KUKA KRL program: MyProgram_058().src

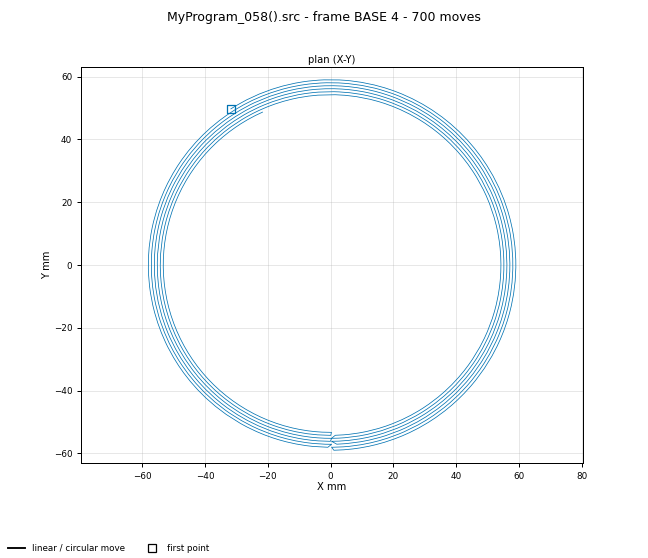
[picture p0: tool path of MyProgram_058().src in frame BASE 4, 700 of 700 moves have a stored position in this frame; points joined in program order, loops and branches not executed]
&ACCESS RVP
&REL 1
&PARAM TEMPLATE = C:\KRC\Roboter\Template\vorgabe
&PARAM EDITMASK = *
DEF MyProgram_058()
; ---- Setting reference (Base) ----
$BASE = BASE_DATA[4]

; --------------------------
; ---- Setting tool (TCP) ----
$TOOL = TOOL_DATA[3]
; --------------------------

$VEL.CP = VEL_APROX_PRINT
Startdeposition()
$VEL.CP = VEL_PRINT
LIN {X -31.7712,Y 49.7386,Z 70,A 115.7642,B 24.8628,C -2.7028,E1 24.9149,E2 -31.8987} C_DIS
LIN {X -30.2288,Y 50.6912,Z 70,A 113.4787,B 24.8635,C -2.6964,E1 24.9204,E2 -29.5909} C_DIS
LIN {X -26.7628,Y 52.603,Z 70,A 109.7045,B 24.8627,C -2.704,E1 24.9297,E2 -25.8244} C_DIS
LIN {X -22.7197,Y 54.4719,Z 70,A 105.0996,B 24.8626,C -2.7051,E1 24.9415,E2 -21.211} C_DIS
LIN {X -18.7389,Y 55.966,Z 70,A 100.782,B 24.8624,C -2.7067,E1 24.9529,E2 -16.8887} C_DIS
LIN {X -15.1635,Y 57.039,Z 70,A 97.4072,B 24.8616,C -2.7151,E1 24.9619,E2 -13.5286} C_DIS
LIN {X -11.2682,Y 57.9341,Z 70,A 94.0177,B 24.8603,C -2.7278,E1 24.9711,E2 -10.1653} C_DIS
LIN {X -8.899,Y 58.3451,Z 70,A 91.7622,B 24.8599,C -2.731,E1 24.9773,E2 -7.9152} C_DIS
LIN {X -6.9633,Y 58.6076,Z 70,A 89.5682,B 24.8604,C -2.7263,E1 24.9834,E2 -5.7084} C_DIS
LIN {X -3.7507,Y 58.9003,Z 70,A 86.8377,B 24.8595,C -2.7356,E1 24.9909,E2 -2.9988} C_DIS
LIN {X -2.0595,Y 58.9836,Z 70,A 84.3436,B 24.8611,C -2.7193,E1 24.998,E2 -0.4657} C_DIS
LIN {X 2.782,Y 58.9546,Z 70,A 80.395,B 24.8595,C -2.7349,E1 25.0089,E2 3.4453} C_DIS
LIN {X 4.6141,Y 58.8391,Z 70,A 78.6103,B 24.8595,C -2.7348,E1 25.0139,E2 5.2294} C_DIS
LIN {X 6.273,Y 58.6855,Z 70,A 76.5349,B 24.8605,C -2.7253,E1 25.0197,E2 7.326} C_DIS
LIN {X 9.7816,Y 58.2035,Z 70,A 73.055,B 24.8607,C -2.7235,E1 25.0293,E2 10.807} C_DIS
LIN {X 13.9156,Y 57.3558,Z 70,A 69.4123,B 24.8599,C -2.7308,E1 25.0392,E2 14.4274} C_DIS
LIN {X 17.2164,Y 56.4534,Z 70,A 65.518,B 24.8614,C -2.7167,E1 25.0497,E2 18.3487} C_DIS
LIN {X 20.0653,Y 55.5043,Z 70,A 63.2005,B 24.8604,C -2.7267,E1 25.0558,E2 20.6377} C_DIS
LIN {X 22.699,Y 54.4806,Z 70,A 59.2086,B 24.8633,C -2.6977,E1 25.0662,E2 24.6892} C_DIS
LIN {X 26.0309,Y 52.9694,Z 70,A 55.6174,B 24.8638,C -2.6926,E1 25.0752,E2 28.2831} C_DIS
LIN {X 29.3497,Y 51.2047,Z 70,A 52.1102,B 24.8641,C -2.6905,E1 25.0837,E2 31.7847} C_DIS
LIN {X 32.329,Y 49.3781,Z 70,A 49.9406,B 24.8619,C -2.7117,E1 25.0887,E2 33.8971} C_DIS
LIN {X 35.5242,Y 47.1314,Z 70,A 46.0197,B 24.8628,C -2.7025,E1 25.0976,E2 37.826} C_DIS
LIN {X 38.2213,Y 44.9718,Z 70,A 41.8696,B 24.8652,C -2.6788,E1 25.1066,E2 42.0164} C_DIS
LIN {X 40.951,Y 42.5011,Z 70,A 37.9748,B 24.8667,C -2.6645,E1 25.1145,E2 45.929} C_DIS
LIN {X 43.5029,Y 39.8852,Z 70,A 34.5086,B 24.8673,C -2.6586,E1 25.121,E2 49.3939} C_DIS
LIN {X 45.8007,Y 37.224,Z 70,A 32.1171,B 24.8658,C -2.6735,E1 25.1252,E2 51.7391} C_DIS
LIN {X 47.9004,Y 34.481,Z 70,A 29.1684,B 24.8657,C -2.6747,E1 25.1302,E2 54.671} C_DIS
LIN {X 49.7604,Y 31.7374,Z 70,A 25.887,B 24.8666,C -2.6651,E1 25.1353,E2 57.9586} C_DIS
LIN {X 51.7267,Y 28.4214,Z 70,A 22.1297,B 24.8676,C -2.655,E1 25.1406,E2 61.7206} C_DIS
LIN {X 53.6143,Y 24.6759,Z 70,A 17.7843,B 24.8694,C -2.6375,E1 25.146,E2 66.0841} C_DIS
LIN {X 55.207,Y 20.8685,Z 70,A 13.7674,B 24.8705,C -2.6259,E1 25.1502,E2 70.1063} C_DIS
LIN {X 56.4433,Y 17.2492,Z 70,A 10.1855,B 24.8713,C -2.618,E1 25.1533,E2 73.6865} C_DIS
LIN {X 57.2283,Y 14.428,Z 70,A 7.3114,B 24.8722,C -2.6088,E1 25.1554,E2 76.566} C_DIS
LIN {X 57.9039,Y 11.4254,Z 70,A 4.541,B 24.8726,C -2.6048,E1 25.157,E2 79.3297} C_DIS
LIN {X 58.3023,Y 9.1755,Z 70,A 1.1429,B 24.876,C -2.5705,E1 25.1585,E2 82.789} C_DIS
LIN {X 58.747,Y 5.6725,Z 70,A -0.9763,B 24.874,C -2.5903,E1 25.1591,E2 84.8487} C_DIS
LIN {X 58.9966,Y 1.6596,Z 70,A -5.4445,B 24.8765,C -2.5648,E1 25.1598,E2 89.3507} C_DIS
LIN {X 59.0156,Y -0.7643,Z 70,A -7.8914,B 24.8774,C -2.5551,E1 25.1598,E2 91.8058} C_DIS
LIN {X 58.8028,Y -5.0655,Z 70,A -11.3027,B 24.877,C -2.56,E1 25.1591,E2 95.1854} C_DIS
LIN {X 58.2932,Y -9.2343,Z 70,A -16.1939,B 24.88,C -2.528,E1 25.1573,E2 100.1234} C_DIS
LIN {X 57.5759,Y -12.9783,Z 70,A -19.3572,B 24.88,C -2.529,E1 25.1555,E2 103.266} C_DIS
LIN {X 57.0238,Y -15.2198,Z 70,A -21.3949,B 24.8801,C -2.5268,E1 25.1541,E2 105.297} C_DIS
LIN {X 56.2334,Y -17.922,Z 70,A -24.511,B 24.8818,C -2.5094,E1 25.1515,E2 108.4366} C_DIS
LIN {X 55.1794,Y -20.9418,Z 70,A -27.4296,B 24.8823,C -2.5043,E1 25.1487,E2 111.3509} C_DIS
LIN {X 54.1381,Y -23.5033,Z 70,A -30.0027,B 24.8828,C -2.4988,E1 25.146,E2 113.9226} C_DIS
LIN {X 53.029,Y -25.9104,Z 70,A -32.634,B 24.8836,C -2.4899,E1 25.1428,E2 116.561} C_DIS
LIN {X 51.3804,Y -29.0427,Z 70,A -35.9802,B 24.8844,C -2.4821,E1 25.1384,E2 119.9081} C_DIS
LIN {X 48.9651,Y -32.951,Z 70,A -40.4263,B 24.8855,C -2.47,E1 25.1317,E2 124.3604} C_DIS
LIN {X 46.171,Y -36.7642,Z 70,A -44.6881,B 24.8859,C -2.4653,E1 25.1246,E2 128.6128} C_DIS
LIN {X 44.7293,Y -38.506,Z 70,A -47.2824,B 24.8873,C -2.4505,E1 25.1199,E2 131.2303} C_DIS
LIN {X 42.5894,Y -40.8593,Z 70,A -50.345,B 24.8879,C -2.4435,E1 25.1141,E2 134.2961} C_DIS
LIN {X 40.4139,Y -43.0121,Z 70,A -53.3512,B 24.8887,C -2.4357,E1 25.108,E2 137.3082} C_DIS
LIN {X 38.5066,Y -44.7285,Z 70,A -55.5701,B 24.8887,C -2.4362,E1 25.1034,E2 139.517} C_DIS
LIN {X 36.3375,Y -46.5083,Z 70,A -59.4128,B 24.8914,C -2.4053,E1 25.0948,E2 143.4186} C_DIS
LIN {X 33.5039,Y -48.5887,Z 70,A -61.8182,B 24.89,C -2.4209,E1 25.0894,E2 145.7788} C_DIS
LIN {X 31.069,Y -50.1807,Z 70,A -64.8964,B 24.891,C -2.4099,E1 25.0821,E2 148.8731} C_DIS
LIN {X 28.1391,Y -51.8798,Z 70,A -68.1417,B 24.8914,C -2.4052,E1 25.0742,E2 152.1201} C_DIS
LIN {X 25.2158,Y -53.3627,Z 70,A -71.046,B 24.8914,C -2.4062,E1 25.067,E2 155.0143} C_DIS
LIN {X 22.836,Y -54.4229,Z 70,A -73.5731,B 24.8917,C -2.4025,E1 25.0605,E2 157.5439} C_DIS
LIN {X 20.2386,Y -55.4412,Z 70,A -76.3101,B 24.8921,C -2.3983,E1 25.0533,E2 160.285} C_DIS
LIN {X 17.1773,Y -56.4656,Z 70,A -79.6955,B 24.8929,C -2.3892,E1 25.0443,E2 163.6858} C_DIS
LIN {X 14.4326,Y -57.2285,Z 70,A -82.0061,B 24.8923,C -2.3961,E1 25.0381,E2 165.9764} C_DIS
LIN {X 12.2163,Y -57.7424,Z 70,A -84.4155,B 24.8928,C -2.3898,E1 25.0315,E2 168.3975} C_DIS
LIN {X 9.3879,Y -58.2693,Z 70,A -86.8704,B 24.8924,C -2.3948,E1 25.0248,E2 170.8379} C_DIS
LIN {X 7.1217,Y -58.5886,Z 70,A -89.4603,B 24.8932,C -2.3856,E1 25.0176,E2 173.4475} C_DIS
LIN {X 4.2204,Y -58.8691,Z 70,A -92.2877,B 24.8933,C -2.3843,E1 25.0097,E2 176.2766} C_DIS
LIN {X 1.0462,Y -59.0104,Z 70,A -95.2132,B 24.8931,C -2.3866,E1 25.0015,E2 179.196} C_DIS
LIN {X 1.0462,Y -59.0104,Z 70,A -95.2132,B 24.8931,C -2.3866,E1 25.0015,E2 179.196} C_DIS
Enddeposition()
LIN {X 0.3368,Y -58.0655,Z 70,A -95.8183,B 24.8915,C -2.4048,E1 25,E2 179.7576} C_DIS
Startdeposition()
$VEL.CP = VEL_PRINT
LIN {X 4.0061,Y -57.93,Z 70,A -91.3397,B 24.8898,C -2.4236,E1 25.0126,E2 175.2355} C_DIS
LIN {X 6.0336,Y -57.754,Z 70,A -88.5797,B 24.8882,C -2.4406,E1 25.0204,E2 172.437} C_DIS
LIN {X 9.6767,Y -57.2564,Z 70,A -84.9689,B 24.888,C -2.4428,E1 25.0303,E2 168.8244} C_DIS
LIN {X 12.7797,Y -56.6453,Z 70,A -82.2927,B 24.8886,C -2.436,E1 25.0376,E2 166.1679} C_DIS
LIN {X 15.542,Y -55.9504,Z 70,A -79.5466,B 24.8885,C -2.4375,E1 25.045,E2 163.4225} C_DIS
LIN {X 18.2311,Y -55.1325,Z 70,A -76.5661,B 24.8878,C -2.4453,E1 25.053,E2 160.4291} C_DIS
LIN {X 21.8468,Y -53.8019,Z 70,A -73.2635,B 24.8883,C -2.4395,E1 25.0615,E2 157.1474} C_DIS
LIN {X 23.4032,Y -53.1438,Z 70,A -70.8909,B 24.8866,C -2.4575,E1 25.0677,E2 154.7378} C_DIS
LIN {X 27.8224,Y -50.9692,Z 70,A -66.6091,B 24.8871,C -2.4526,E1 25.0783,E2 150.4795} C_DIS
LIN {X 30.5558,Y -49.3795,Z 70,A -63.1211,B 24.8858,C -2.4665,E1 25.0867,E2 146.9693} C_DIS
LIN {X 32.792,Y -47.9238,Z 70,A -60.5015,B 24.8854,C -2.4714,E1 25.0927,E2 144.3471} C_DIS
LIN {X 36.1303,Y -45.4594,Z 70,A -56.8016,B 24.8854,C -2.471,E1 25.1009,E2 140.6615} C_DIS
LIN {X 37.9818,Y -43.923,Z 70,A -54.0281,B 24.8841,C -2.4854,E1 25.1069,E2 137.8648} C_DIS
LIN {X 40.8451,Y -41.2748,Z 70,A -50.3062,B 24.8835,C -2.4915,E1 25.1144,E2 134.1438} C_DIS
LIN {X 43.5271,Y -38.435,Z 70,A -46.9008,B 24.8835,C -2.4907,E1 25.1208,E2 130.7553} C_DIS
LIN {X 45.0965,Y -36.5819,Z 70,A -43.953,B 24.8818,C -2.5096,E1 25.1261,E2 127.7763} C_DIS
LIN {X 47.5483,Y -33.3337,Z 70,A -40.6437,B 24.8823,C -2.504,E1 25.1315,E2 124.4963} C_DIS
LIN {X 48.9925,Y -31.1723,Z 70,A -37.4768,B 24.8803,C -2.5251,E1 25.1364,E2 121.2953} C_DIS
LIN {X 50.6871,Y -28.3328,Z 70,A -33.9859,B 24.8789,C -2.5398,E1 25.1412,E2 117.7878} C_DIS
LIN {X 52.8545,Y -24.0493,Z 70,A -30.051,B 24.8794,C -2.5348,E1 25.146,E2 113.8857} C_DIS
LIN {X 53.5161,Y -22.5379,Z 70,A -27.9151,B 24.8778,C -2.5516,E1 25.1484,E2 111.7218} C_DIS
LIN {X 54.8862,Y -18.9604,Z 70,A -24.4347,B 24.8774,C -2.556,E1 25.1517,E2 108.2504} C_DIS
LIN {X 55.7308,Y -16.3106,Z 70,A -21.7341,B 24.8766,C -2.5635,E1 25.1539,E2 105.5476} C_DIS
LIN {X 56.4512,Y -13.6094,Z 70,A -19.2381,B 24.8764,C -2.5659,E1 25.1556,E2 103.0603} C_DIS
LIN {X 57.3258,Y -9.2615,Z 70,A -14.9406,B 24.8753,C -2.5777,E1 25.1579,E2 98.7599} C_DIS
LIN {X 57.803,Y -5.5483,Z 70,A -11.1473,B 24.8739,C -2.5917,E1 25.1592,E2 94.956} C_DIS
LIN {X 58.0553,Y -1.2392,Z 70,A -6.9847,B 24.8728,C -2.6029,E1 25.1598,E2 90.7917} C_DIS
LIN {X 58.0291,Y 2.1446,Z 70,A -2.8172,B 24.8698,C -2.633,E1 25.1595,E2 86.5777} C_DIS
LIN {X 57.6965,Y 6.5634,Z 70,A 1.1575,B 24.8694,C -2.6372,E1 25.1584,E2 82.6167} C_DIS
LIN {X 57.2137,Y 9.9317,Z 70,A 4.1816,B 24.8692,C -2.6397,E1 25.1571,E2 79.6045} C_DIS
LIN {X 56.887,Y 11.653,Z 70,A 6.4002,B 24.8675,C -2.6565,E1 25.1559,E2 77.3591} C_DIS
LIN {X 55.7905,Y 16.1067,Z 70,A 10.1188,B 24.868,C -2.6511,E1 25.1533,E2 73.6746} C_DIS
LIN {X 54.7562,Y 19.3311,Z 70,A 13.5403,B 24.8669,C -2.6628,E1 25.1503,E2 70.2449} C_DIS
LIN {X 54.0939,Y 21.1138,Z 70,A 15.9706,B 24.865,C -2.6811,E1 25.1478,E2 67.7848} C_DIS
LIN {X 52.902,Y 23.9439,Z 70,A 19.526,B 24.8629,C -2.7018,E1 25.1437,E2 64.1997} C_DIS
LIN {X 51.104,Y 27.5739,Z 70,A 23.5816,B 24.8617,C -2.7139,E1 25.1384,E2 60.1368} C_DIS
LIN {X 49.4059,Y 30.5134,Z 70,A 25.7534,B 24.8636,C -2.6954,E1 25.1354,E2 58.02} C_DIS
LIN {X 47.5937,Y 33.2683,Z 70,A 29.4558,B 24.8617,C -2.7138,E1 25.1295,E2 54.2923} C_DIS
LIN {X 45.5686,Y 35.992,Z 70,A 32.214,B 24.8622,C -2.7083,E1 25.1249,E2 51.5601} C_DIS
LIN {X 43.7453,Y 38.1873,Z 70,A 35.3315,B 24.8609,C -2.7216,E1 25.1193,E2 48.4256} C_DIS
LIN {X 42.43,Y 39.6442,Z 70,A 38.0863,B 24.8586,C -2.7442,E1 25.1139,E2 45.6291} C_DIS
LIN {X 39.5187,Y 42.5478,Z 70,A 41.7521,B 24.8586,C -2.7436,E1 25.1065,E2 41.98} C_DIS
LIN {X 36.5071,Y 45.157,Z 70,A 45.3575,B 24.8586,C -2.7437,E1 25.0988,E2 38.3882} C_DIS
LIN {X 34.84,Y 46.4554,Z 70,A 47.519,B 24.8581,C -2.749,E1 25.094,E2 36.2219} C_DIS
LIN {X 31.8583,Y 48.5488,Z 70,A 50.6064,B 24.8586,C -2.7437,E1 25.087,E2 33.1575} C_DIS
LIN {X 28.6355,Y 50.5178,Z 70,A 55.493,B 24.8554,C -2.7743,E1 25.075,E2 28.2133} C_DIS
LIN {X 25.7741,Y 52.0348,Z 70,A 57.857,B 24.8569,C -2.7603,E1 25.0693,E2 25.889} C_DIS
LIN {X 21.8175,Y 53.8138,Z 70,A 61.9803,B 24.8568,C -2.7615,E1 25.0587,E2 21.7727} C_DIS
LIN {X 19.5455,Y 54.6808,Z 70,A 64.7617,B 24.8557,C -2.7717,E1 25.0514,E2 18.9729} C_DIS
LIN {X 15.6188,Y 55.928,Z 70,A 68.2352,B 24.8567,C -2.7623,E1 25.0422,E2 15.5279} C_DIS
LIN {X 14.1219,Y 56.3253,Z 70,A 70.4889,B 24.855,C -2.7783,E1 25.036,E2 13.2396} C_DIS
LIN {X 10.0125,Y 57.1992,Z 70,A 74.5226,B 24.855,C -2.7776,E1 25.0249,E2 9.2122} C_DIS
LIN {X 5.3929,Y 57.8173,Z 70,A 78.9116,B 24.8554,C -2.7741,E1 25.0128,E2 4.8347} C_DIS
LIN {X 2.5862,Y 58.0107,Z 70,A 81.7846,B 24.8553,C -2.776,E1 25.0048,E2 1.9583} C_DIS
LIN {X -1.2933,Y 58.0543,Z 70,A 85.1594,B 24.8563,C -2.7662,E1 24.9954,E2 -1.393} C_DIS
LIN {X -3.1849,Y 57.9809,Z 70,A 87.3647,B 24.8556,C -2.7722,E1 24.9892,E2 -3.6132} C_DIS
LIN {X -6.7659,Y 57.6728,Z 70,A 90.7348,B 24.8562,C -2.7669,E1 24.9799,E2 -6.9726} C_DIS
LIN {X -9.6106,Y 57.2675,Z 70,A 93.6963,B 24.8562,C -2.7675,E1 24.9717,E2 -9.938} C_DIS
LIN {X -12.5839,Y 56.6888,Z 70,A 96.8429,B 24.8561,C -2.768,E1 24.9631,E2 -13.0897} C_DIS
LIN {X -15.2568,Y 56.0283,Z 70,A 99.8798,B 24.8557,C -2.7715,E1 24.9549,E2 -16.1394} C_DIS
LIN {X -18.9545,Y 54.8884,Z 70,A 103.0395,B 24.8575,C -2.7545,E1 24.9466,E2 -19.2644} C_DIS
LIN {X -21.8103,Y 53.8168,Z 70,A 106.3993,B 24.8572,C -2.7571,E1 24.9378,E2 -22.6376} C_DIS
LIN {X -24.9043,Y 52.4574,Z 70,A 109.1655,B 24.8588,C -2.7416,E1 24.9308,E2 -25.3736} C_DIS
LIN {X -27.6387,Y 51.0689,Z 70,A 112.9934,B 24.8578,C -2.7515,E1 24.9213,E2 -29.2356} C_DIS
LIN {X -30.7549,Y 49.2551,Z 70,A 116.2345,B 24.8591,C -2.7393,E1 24.9136,E2 -32.4576} C_DIS
LIN {X -33.0294,Y 47.7599,Z 70,A 118.7367,B 24.8599,C -2.7308,E1 24.9078,E2 -34.9478} C_DIS
LIN {X -35.3908,Y 46.0372,Z 70,A 121.9748,B 24.8599,C -2.7313,E1 24.9005,E2 -38.1987} C_DIS
LIN {X -38.288,Y 43.6574,Z 70,A 125.3415,B 24.8613,C -2.7172,E1 24.8934,E2 -41.5448} C_DIS
LIN {X -40.5568,Y 41.5579,Z 70,A 128.7411,B 24.8614,C -2.7164,E1 24.8865,E2 -44.9565} C_DIS
LIN {X -42.9807,Y 39.0465,Z 70,A 132.2773,B 24.8621,C -2.7097,E1 24.8797,E2 -48.492} C_DIS
LIN {X -45.4039,Y 36.2004,Z 70,A 136.0486,B 24.8629,C -2.7017,E1 24.8731,E2 -52.2617} C_DIS
LIN {X -47.4887,Y 33.4194,Z 70,A 139.2387,B 24.8643,C -2.6883,E1 24.8679,E2 -55.4354} C_DIS
LIN {X -48.7906,Y 31.4868,Z 70,A 141.2399,B 24.8654,C -2.6769,E1 24.8648,E2 -57.4192} C_DIS
LIN {X -50.2196,Y 29.1544,Z 70,A 144.3862,B 24.8654,C -2.677,E1 24.8603,E2 -60.5821} C_DIS
LIN {X -51.8909,Y 26.063,Z 70,A 147.9848,B 24.8662,C -2.6693,E1 24.8557,E2 -64.1814} C_DIS
LIN {X -53.0729,Y 23.5646,Z 70,A 150.1524,B 24.868,C -2.6516,E1 24.8532,E2 -66.3187} C_DIS
LIN {X -54.2492,Y 20.7117,Z 70,A 154.0378,B 24.8674,C -2.6569,E1 24.8491,E2 -70.2385} C_DIS
LIN {X -55.4296,Y 17.3061,Z 70,A 157.3705,B 24.8689,C -2.6422,E1 24.8463,E2 -73.555} C_DIS
LIN {X -56.4076,Y 13.7882,Z 70,A 160.5004,B 24.8708,C -2.6229,E1 24.8441,E2 -76.6572} C_DIS
LIN {X -56.8516,Y 11.824,Z 70,A 162.5908,B 24.8713,C -2.6185,E1 24.8428,E2 -78.7492} C_DIS
LIN {X -57.2638,Y 9.6323,Z 70,A 165.1916,B 24.8713,C -2.6185,E1 24.8416,E2 -81.3653} C_DIS
LIN {X -57.8002,Y 5.5788,Z 70,A 169.254,B 24.8725,C -2.6061,E1 24.8403,E2 -85.4227} C_DIS
LIN {X -58.0131,Y 2.53,Z 70,A 172.2094,B 24.8735,C -2.5956,E1 24.8398,E2 -88.3706} C_DIS
LIN {X -58.0572,Y -1.1344,Z 70,A 175.4406,B 24.8753,C -2.5776,E1 24.8398,E2 -91.5783} C_DIS
LIN {X -57.982,Y -3.1649,Z 70,A 177.7382,B 24.8753,C -2.5763,E1 24.8401,E2 -93.8867} C_DIS
LIN {X -57.6791,Y -6.7118,Z 70,A -178.9542,B 24.8768,C -2.5619,E1 24.841,E2 -97.1795} C_DIS
LIN {X -57.3992,Y -8.7866,Z 70,A -176.0673,B 24.876,C -2.5697,E1 24.8422,E2 -100.1023} C_DIS
LIN {X -56.6399,Y -12.8033,Z 70,A -173.0126,B 24.8788,C -2.5405,E1 24.8439,E2 -103.1052} C_DIS
LIN {X -56.0504,Y -15.1747,Z 70,A -170.1321,B 24.8788,C -2.5413,E1 24.8459,E2 -106.0045} C_DIS
LIN {X -55.0664,Y -18.4267,Z 70,A -166.2436,B 24.8788,C -2.5408,E1 24.8493,E2 -109.9141} C_DIS
LIN {X -53.9363,Y -21.5135,Z 70,A -163.3509,B 24.8803,C -2.5254,E1 24.8522,E2 -112.7862} C_DIS
LIN {X -52.5831,Y -24.6365,Z 70,A -160.4693,B 24.882,C -2.5077,E1 24.8554,E2 -115.6413} C_DIS
LIN {X -51.8846,Y -26.0766,Z 70,A -158.2162,B 24.8812,C -2.5152,E1 24.8583,E2 -117.9245} C_DIS
LIN {X -50.001,Y -29.5262,Z 70,A -154.846,B 24.8831,C -2.496,E1 24.8629,E2 -121.2665} C_DIS
LIN {X -48.3842,Y -32.1081,Z 70,A -151.25,B 24.8828,C -2.4989,E1 24.8684,E2 -124.8875} C_DIS
LIN {X -46.7722,Y -34.4137,Z 70,A -148.7066,B 24.8838,C -2.488,E1 24.8725,E2 -127.4173} C_DIS
LIN {X -44.7315,Y -37.0274,Z 70,A -145.6423,B 24.8849,C -2.4767,E1 24.8779,E2 -130.4687} C_DIS
LIN {X -42.2486,Y -39.837,Z 70,A -141.3411,B 24.8846,C -2.4796,E1 24.886,E2 -134.7959} C_DIS
LIN {X -39.6939,Y -42.3832,Z 70,A -137.4422,B 24.8846,C -2.4787,E1 24.8939,E2 -138.7089} C_DIS
LIN {X -36.69,Y -45.0089,Z 70,A -133.4944,B 24.8853,C -2.4717,E1 24.9024,E2 -142.6549} C_DIS
LIN {X -33.2602,Y -47.5994,Z 70,A -129.5351,B 24.8865,C -2.4593,E1 24.9114,E2 -146.5985} C_DIS
LIN {X -28.6805,Y -50.4919,Z 70,A -124.9588,B 24.8886,C -2.4369,E1 24.9222,E2 -151.1355} C_DIS
LIN {X -26.639,Y -51.5979,Z 70,A -121.9747,B 24.8876,C -2.4473,E1 24.9296,E2 -154.1526} C_DIS
LIN {X -23.6199,Y -53.048,Z 70,A -119.1743,B 24.8888,C -2.4338,E1 24.9367,E2 -156.9279} C_DIS
LIN {X -21.0188,Y -54.131,Z 70,A -116.2578,B 24.8888,C -2.4338,E1 24.9442,E2 -159.8508} C_DIS
LIN {X -18.4558,Y -55.0574,Z 70,A -113.659,B 24.8892,C -2.4298,E1 24.9511,E2 -162.4452} C_DIS
LIN {X -16.2663,Y -55.744,Z 70,A -111.49,B 24.8895,C -2.4264,E1 24.9569,E2 -164.6096} C_DIS
LIN {X -14.0521,Y -56.3432,Z 70,A -109.1453,B 24.8895,C -2.4267,E1 24.9632,E2 -166.9585} C_DIS
LIN {X -11.0255,Y -57.012,Z 70,A -105.6761,B 24.8888,C -2.4337,E1 24.9728,E2 -170.4484} C_DIS
LIN {X -7.8663,Y -57.5333,Z 70,A -102.9456,B 24.8897,C -2.4242,E1 24.9802,E2 -173.1587} C_DIS
LIN {X -5.7466,Y -57.784,Z 70,A -100.2879,B 24.8887,C -2.4353,E1 24.9877,E2 -175.8443} C_DIS
LIN {X -0.8759,Y -58.0619,Z 70,A -95.9188,B 24.8895,C -2.4266,E1 24.9998,E2 -180.1935} C_DIS
LIN {X -0.8759,Y -58.0619,Z 70,A -95.9188,B 24.8895,C -2.4266,E1 24.9998,E2 -180.1935} C_DIS
Enddeposition()
LIN {X 0.3217,Y -57.1143,Z 70,A -94.8754,B 24.8882,C -2.4403,E1 25.0029,E2 -181.2696} C_DIS
Startdeposition()
$VEL.CP = VEL_PRINT
LIN {X -1.6753,Y -57.0923,Z 70,A -98.3895,B 24.891,C -2.4097,E1 24.9928,E2 -177.6824} C_DIS
LIN {X -5.5522,Y -56.8472,Z 70,A -101.9141,B 24.8904,C -2.417,E1 24.9831,E2 -174.1738} C_DIS
LIN {X -8.11,Y -56.5382,Z 70,A -104.2999,B 24.89,C -2.4214,E1 24.9765,E2 -171.7967} C_DIS
LIN {X -11.1706,Y -56.0141,Z 70,A -107.9954,B 24.8909,C -2.4113,E1 24.9663,E2 -168.0732} C_DIS
LIN {X -14.0088,Y -55.3725,Z 70,A -110.4419,B 24.8899,C -2.4218,E1 24.9597,E2 -165.6484} C_DIS
LIN {X -16.4763,Y -54.6884,Z 70,A -113.2493,B 24.8902,C -2.4189,E1 24.9521,E2 -162.8297} C_DIS
LIN {X -19.2701,Y -53.769,Z 70,A -116.3655,B 24.8902,C -2.4182,E1 24.9439,E2 -159.7057} C_DIS
LIN {X -22.8472,Y -52.3483,Z 70,A -119.8469,B 24.8893,C -2.4291,E1 24.9349,E2 -156.2425} C_DIS
LIN {X -24.9522,Y -51.3783,Z 70,A -122.9194,B 24.8903,C -2.4181,E1 24.9271,E2 -153.1358} C_DIS
LIN {X -28.4494,Y -49.5275,Z 70,A -126.7876,B 24.8896,C -2.4252,E1 24.9177,E2 -149.2735} C_DIS
LIN {X -32.168,Y -47.1967,Z 70,A -130.4275,B 24.8877,C -2.4457,E1 24.9092,E2 -145.6706} C_DIS
LIN {X -33.522,Y -46.2459,Z 70,A -133.1182,B 24.8892,C -2.43,E1 24.903,E2 -142.9332} C_DIS
LIN {X -36.8731,Y -43.6207,Z 70,A -137.4028,B 24.8885,C -2.4376,E1 24.8938,E2 -138.6504} C_DIS
LIN {X -40.1335,Y -40.6403,Z 70,A -141.4744,B 24.8871,C -2.4528,E1 24.8856,E2 -134.5982} C_DIS
LIN {X -42.9586,Y -37.6417,Z 70,A -145.4584,B 24.886,C -2.4644,E1 24.8781,E2 -130.6242} C_DIS
LIN {X -45.3182,Y -34.7651,Z 70,A -149.0744,B 24.885,C -2.4751,E1 24.8719,E2 -127.0168} C_DIS
LIN {X -47.3419,Y -31.9543,Z 70,A -152.4104,B 24.884,C -2.4859,E1 24.8665,E2 -123.6903} C_DIS
LIN {X -48.511,Y -30.1502,Z 70,A -154.7657,B 24.8838,C -2.4881,E1 24.863,E2 -121.3282} C_DIS
LIN {X -50.1157,Y -27.4004,Z 70,A -158.1128,B 24.8833,C -2.4939,E1 24.8584,E2 -117.9775} C_DIS
LIN {X -51.4173,Y -24.8721,Z 70,A -160.6434,B 24.882,C -2.5071,E1 24.8552,E2 -115.4647} C_DIS
LIN {X -52.8836,Y -21.5792,Z 70,A -164.253,B 24.8811,C -2.5173,E1 24.8512,E2 -111.8597} C_DIS
LIN {X -54.1577,Y -18.1463,Z 70,A -167.902,B 24.88,C -2.5283,E1 24.8478,E2 -108.2163} C_DIS
LIN {X -54.7147,Y -16.3909,Z 70,A -170.1922,B 24.8802,C -2.5265,E1 24.8459,E2 -105.9085} C_DIS
LIN {X -55.712,Y -12.5929,Z 70,A -173.6496,B 24.8783,C -2.5462,E1 24.8435,E2 -102.4781} C_DIS
LIN {X -56.1934,Y -10.2262,Z 70,A -176.5738,B 24.8783,C -2.5454,E1 24.842,E2 -99.5348} C_DIS
LIN {X -56.6922,Y -6.9596,Z 70,A -179.8253,B 24.8773,C -2.5567,E1 24.8407,E2 -96.2907} C_DIS
LIN {X -56.9947,Y -3.736,Z 70,A 177.283,B 24.8757,C -2.5726,E1 24.8401,E2 -93.4198} C_DIS
LIN {X -57.0847,Y -1.9147,Z 70,A 174.667,B 24.8764,C -2.5656,E1 24.8398,E2 -90.7713} C_DIS
LIN {X -57.0521,Y 2.7317,Z 70,A 170.6679,B 24.874,C -2.591,E1 24.84,E2 -86.8089} C_DIS
LIN {X -56.9354,Y 4.5496,Z 70,A 168.7831,B 24.8735,C -2.5959,E1 24.8404,E2 -84.9244} C_DIS
LIN {X -56.7303,Y 6.6343,Z 70,A 166.4728,B 24.8732,C -2.5991,E1 24.8411,E2 -82.608} C_DIS
LIN {X -56.3312,Y 9.4407,Z 70,A 163.9146,B 24.8718,C -2.6127,E1 24.8422,E2 -80.0669} C_DIS
LIN {X -56.0575,Y 10.9505,Z 70,A 162.0738,B 24.8718,C -2.6126,E1 24.8431,E2 -78.215} C_DIS
LIN {X -55.475,Y 13.5966,Z 70,A 159.2999,B 24.8711,C -2.6201,E1 24.8449,E2 -75.4429} C_DIS
LIN {X -54.692,Y 16.4675,Z 70,A 156.3825,B 24.8701,C -2.6305,E1 24.8471,E2 -72.5332} C_DIS
LIN {X -53.5452,Y 19.8799,Z 70,A 152.7682,B 24.869,C -2.6414,E1 24.8504,E2 -68.9246} C_DIS
LIN {X -52.6274,Y 22.1968,Z 70,A 150.2278,B 24.8683,C -2.6482,E1 24.8531,E2 -66.3864} C_DIS
LIN {X -51.6026,Y 24.4848,Z 70,A 147.6106,B 24.8677,C -2.6539,E1 24.8562,E2 -63.7685} C_DIS
LIN {X -50.3353,Y 26.9957,Z 70,A 144.3789,B 24.8677,C -2.6553,E1 24.8604,E2 -60.5229} C_DIS
LIN {X -47.9485,Y 31.0375,Z 70,A 140.3994,B 24.8651,C -2.6806,E1 24.8661,E2 -56.5833} C_DIS
LIN {X -46.9904,Y 32.4694,Z 70,A 138.1496,B 24.8655,C -2.6766,E1 24.8697,E2 -54.3128} C_DIS
LIN {X -44.6391,Y 35.6337,Z 70,A 133.5561,B 24.8655,C -2.6763,E1 24.8776,E2 -49.697} C_DIS
LIN {X -41.9452,Y 38.7682,Z 70,A 130.239,B 24.863,C -2.7005,E1 24.8836,E2 -46.4227} C_DIS
LIN {X -40.251,Y 40.5243,Z 70,A 127.7415,B 24.8625,C -2.7055,E1 24.8885,E2 -43.9265} C_DIS
LIN {X -37.922,Y 42.7119,Z 70,A 124.8382,B 24.8613,C -2.7179,E1 24.8945,E2 -41.0412} C_DIS
LIN {X -36.0728,Y 44.2844,Z 70,A 121.9721,B 24.8615,C -2.7158,E1 24.9006,E2 -38.159} C_DIS
LIN {X -34.1636,Y 45.7735,Z 70,A 119.7642,B 24.8606,C -2.7246,E1 24.9055,E2 -35.9642} C_DIS
LIN {X -32.2973,Y 47.1083,Z 70,A 116.9257,B 24.8611,C -2.7199,E1 24.9121,E2 -33.1046} C_DIS
LIN {X -28.9029,Y 49.2645,Z 70,A 113.029,B 24.8601,C -2.7295,E1 24.9213,E2 -29.2189} C_DIS
LIN {X -25.5964,Y 51.061,Z 70,A 109.711,B 24.8586,C -2.7438,E1 24.9294,E2 -25.9258} C_DIS
LIN {X -24.2242,Y 51.7256,Z 70,A 107.3219,B 24.8599,C -2.7309,E1 24.9356,E2 -23.4999} C_DIS
LIN {X -19.252,Y 53.7755,Z 70,A 101.9478,B 24.8592,C -2.7384,E1 24.9496,E2 -18.1321} C_DIS
LIN {X -15.0599,Y 55.0959,Z 70,A 98.327,B 24.8572,C -2.7575,E1 24.9591,E2 -14.5508} C_DIS
LIN {X -13.439,Y 55.5134,Z 70,A 96.3859,B 24.8575,C -2.7543,E1 24.9644,E2 -12.5993} C_DIS
LIN {X -10.8751,Y 56.072,Z 70,A 93.5266,B 24.8577,C -2.7522,E1 24.9723,E2 -9.7318} C_DIS
LIN {X -6.992,Y 56.6884,Z 70,A 89.8684,B 24.8569,C -2.7601,E1 24.9823,E2 -6.0893} C_DIS
LIN {X -4.5327,Y 56.9367,Z 70,A 87.4552,B 24.8567,C -2.7626,E1 24.989,E2 -3.6808} C_DIS
LIN {X -1.944,Y 57.0841,Z 70,A 84.6806,B 24.8569,C -2.7601,E1 24.9968,E2 -0.8998} C_DIS
LIN {X 0.909,Y 57.1098,Z 70,A 81.7964,B 24.8569,C -2.7602,E1 25.0048,E2 1.984} C_DIS
LIN {X 3.3817,Y 57.0171,Z 70,A 79.4695,B 24.8566,C -2.7633,E1 25.0113,E2 4.3028} C_DIS
LIN {X 5.6615,Y 56.8363,Z 70,A 77.1417,B 24.8566,C -2.7625,E1 25.0178,E2 6.6313} C_DIS
LIN {X 8.6238,Y 56.4622,Z 70,A 73.9556,B 24.8571,C -2.758,E1 25.0266,E2 9.8252} C_DIS
LIN {X 11.722,Y 55.9016,Z 70,A 70.7921,B 24.8573,C -2.7566,E1 25.0353,E2 12.9883} C_DIS
LIN {X 14.1408,Y 55.3388,Z 70,A 68.6854,B 24.8566,C -2.7629,E1 25.041,E2 15.077} C_DIS
LIN {X 16.245,Y 54.758,Z 70,A 66.3068,B 24.8572,C -2.7576,E1 25.0474,E2 17.4642} C_DIS
LIN {X 18.5443,Y 54.0231,Z 70,A 63.8601,B 24.8574,C -2.7551,E1 25.0538,E2 19.912} C_DIS
LIN {X 21.02,Y 53.1085,Z 70,A 61.0514,B 24.858,C -2.7494,E1 25.0612,E2 22.7284} C_DIS
LIN {X 25.3508,Y 51.1827,Z 70,A 57.0895,B 24.8569,C -2.7604,E1 25.0712,E2 26.6542} C_DIS
LIN {X 27.9188,Y 49.8285,Z 70,A 53.0381,B 24.8597,C -2.7328,E1 25.0813,E2 30.7593} C_DIS
LIN {X 31.1722,Y 47.8615,Z 70,A 49.698,B 24.8593,C -2.737,E1 25.0891,E2 34.0789} C_DIS
LIN {X 33.6583,Y 46.1462,Z 70,A 46.7534,B 24.8596,C -2.7337,E1 25.0958,E2 37.021} C_DIS
LIN {X 36.0869,Y 44.273,Z 70,A 43.6021,B 24.8604,C -2.7266,E1 25.1027,E2 40.1774} C_DIS
LIN {X 38.6321,Y 42.0702,Z 70,A 40.356,B 24.8608,C -2.7229,E1 25.1095,E2 43.4195} C_DIS
LIN {X 41.3505,Y 39.4017,Z 70,A 36.5769,B 24.8615,C -2.7158,E1 25.117,E2 47.1993} C_DIS
LIN {X 43.9326,Y 36.5001,Z 70,A 32.8699,B 24.862,C -2.7112,E1 25.1238,E2 50.9005} C_DIS
LIN {X 45.0415,Y 35.1236,Z 70,A 30.629,B 24.8634,C -2.6968,E1 25.1277,E2 53.165} C_DIS
LIN {X 47.0762,Y 32.3449,Z 70,A 27.132,B 24.8644,C -2.6874,E1 25.1333,E2 56.6672} C_DIS
LIN {X 48.7104,Y 29.8273,Z 70,A 23.7598,B 24.866,C -2.6717,E1 25.1383,E2 60.0594} C_DIS
LIN {X 51.2874,Y 25.1376,Z 70,A 18.755,B 24.8666,C -2.6653,E1 25.1448,E2 65.053} C_DIS
LIN {X 52.3557,Y 22.8303,Z 70,A 16.4453,B 24.8668,C -2.6635,E1 25.1474,E2 67.3543} C_DIS
LIN {X 53.7973,Y 19.1905,Z 70,A 12.6312,B 24.8677,C -2.6547,E1 25.1512,E2 71.1679} C_DIS
LIN {X 54.6598,Y 16.575,Z 70,A 10.1111,B 24.8679,C -2.6521,E1 25.1533,E2 73.68} C_DIS
LIN {X 55.4234,Y 13.8079,Z 70,A 6.7547,B 24.8699,C -2.6327,E1 25.1557,E2 77.063} C_DIS
LIN {X 56.0433,Y 11.0241,Z 70,A 4.3528,B 24.8697,C -2.6343,E1 25.1571,E2 79.4469} C_DIS
LIN {X 56.4592,Y 8.643,Z 70,A 1.8552,B 24.8706,C -2.6252,E1 25.1582,E2 81.9515} C_DIS
LIN {X 56.9311,Y 4.6027,Z 70,A -2.5882,B 24.8727,C -2.6043,E1 25.1595,E2 86.418} C_DIS
LIN {X 57.1153,Y 0.5249,Z 70,A -6.1775,B 24.8727,C -2.6029,E1 25.1598,E2 89.9893} C_DIS
LIN {X 57.0817,Y -2.0223,Z 70,A -9.2435,B 24.8747,C -2.5832,E1 25.1595,E2 93.0836} C_DIS
LIN {X 56.8278,Y -5.7427,Z 70,A -13.1144,B 24.8762,C -2.5684,E1 25.1586,E2 96.9665} C_DIS
LIN {X 56.3932,Y -9.0699,Z 70,A -17.0409,B 24.8784,C -2.5452,E1 25.1569,E2 100.9249} C_DIS
LIN {X 55.6853,Y -12.7084,Z 70,A -19.1599,B 24.876,C -2.5698,E1 25.1557,E2 102.9733} C_DIS
LIN {X 55.3353,Y -14.1543,Z 70,A -21.5989,B 24.8785,C -2.5436,E1 25.154,E2 105.4602} C_DIS
LIN {X 54.389,Y -17.4411,Z 70,A -24.2849,B 24.8779,C -2.5499,E1 25.1518,E2 108.1159} C_DIS
LIN {X 53.3253,Y -20.4649,Z 70,A -28.2362,B 24.8805,C -2.5235,E1 25.1479,E2 112.1077} C_DIS
LIN {X 52.1008,Y -23.4061,Z 70,A -31.2725,B 24.881,C -2.5175,E1 25.1445,E2 115.1414} C_DIS
LIN {X 49.8399,Y -27.8985,Z 70,A -35.9714,B 24.8817,C -2.5107,E1 25.1385,E2 119.8316} C_DIS
LIN {X 48.0818,Y -30.8298,Z 70,A -39.6105,B 24.883,C -2.4964,E1 25.1331,E2 123.4861} C_DIS
LIN {X 45.476,Y -34.5597,Z 70,A -44.3078,B 24.8844,C -2.4812,E1 25.1253,E2 128.1966} C_DIS
LIN {X 43.3292,Y -37.2151,Z 70,A -47.8088,B 24.8854,C -2.4708,E1 25.119,E2 131.7063} C_DIS
LIN {X 40.1677,Y -40.6065,Z 70,A -52.2194,B 24.886,C -2.4648,E1 25.1105,E2 136.1121} C_DIS
LIN {X 36.7463,Y -43.728,Z 70,A -56.3797,B 24.886,C -2.465,E1 25.1018,E2 140.2555} C_DIS
LIN {X 34.02,Y -45.8813,Z 70,A -60.4545,B 24.8878,C -2.4448,E1 25.0927,E2 144.3631} C_DIS
LIN {X 30.2725,Y -48.4346,Z 70,A -64.7283,B 24.8881,C -2.442,E1 25.0827,E2 148.6295} C_DIS
LIN {X 27.6275,Y -49.9912,Z 70,A -68.4137,B 24.8897,C -2.4238,E1 25.0737,E2 152.3473} C_DIS
LIN {X 23.8797,Y -51.886,Z 70,A -71.705,B 24.8886,C -2.4366,E1 25.0655,E2 155.5995} C_DIS
LIN {X 22.0826,Y -52.6754,Z 70,A -74.2462,B 24.8899,C -2.4217,E1 25.0589,E2 158.17} C_DIS
LIN {X 17.5486,Y -54.3542,Z 70,A -78.2924,B 24.889,C -2.4324,E1 25.0483,E2 162.1826} C_DIS
LIN {X 15.7517,Y -54.9022,Z 70,A -80.9348,B 24.8906,C -2.4146,E1 25.0411,E2 164.8628} C_DIS
LIN {X 12.341,Y -55.768,Z 70,A -84.4523,B 24.8909,C -2.4116,E1 25.0315,E2 168.3827} C_DIS
LIN {X 9.5701,Y -56.3096,Z 70,A -86.7919,B 24.8901,C -2.4194,E1 25.0252,E2 170.7012} C_DIS
LIN {X 4.9251,Y -56.9037,Z 70,A -91.3339,B 24.8901,C -2.4198,E1 25.0126,E2 175.2389} C_DIS
LIN {X 1.9775,Y -57.0831,Z 70,A -93.9877,B 24.8897,C -2.4248,E1 25.0052,E2 177.8798} C_DIS
LIN {X 1.9775,Y -57.0831,Z 70,A -93.9877,B 24.8897,C -2.4248,E1 25.0052,E2 177.8798} C_DIS
Enddeposition()
LIN {X 0.3099,Y -56.1615,Z 70,A -95.1001,B 24.8872,C -2.4521,E1 25.0023,E2 178.9272} C_DIS
Startdeposition()
$VEL.CP = VEL_PRINT
LIN {X 2.6789,Y -56.1021,Z 70,A -92.4847,B 24.8867,C -2.4568,E1 25.0096,E2 176.3012} C_DIS
LIN {X 5.8531,Y -55.8596,Z 70,A -88.772,B 24.8857,C -2.4679,E1 25.02,E2 172.5642} C_DIS
LIN {X 9.423,Y -55.3696,Z 70,A -85.7766,B 24.8867,C -2.4565,E1 25.0282,E2 169.5987} C_DIS
LIN {X 12.0412,Y -54.8596,Z 70,A -82.7636,B 24.886,C -2.4649,E1 25.0365,E2 166.5696} C_DIS
LIN {X 14.7486,Y -54.1943,Z 70,A -79.98,B 24.8858,C -2.4665,E1 25.044,E2 163.7865} C_DIS
LIN {X 16.8646,Y -53.5743,Z 70,A -77.2278,B 24.8846,C -2.4797,E1 25.0514,E2 161.008} C_DIS
LIN {X 21.2307,Y -51.9983,Z 70,A -72.9884,B 24.885,C -2.4755,E1 25.0624,E2 156.7878} C_DIS
LIN {X 24.6249,Y -50.4805,Z 70,A -68.5583,B 24.8832,C -2.495,E1 25.0737,E2 152.3227} C_DIS
LIN {X 28.1829,Y -48.5833,Z 70,A -65.3462,B 24.8843,C -2.4826,E1 25.0815,E2 149.1493} C_DIS
LIN {X 30.3057,Y -47.2876,Z 70,A -62.5744,B 24.8834,C -2.4924,E1 25.0881,E2 146.3631} C_DIS
LIN {X 33.2374,Y -45.2751,Z 70,A -58.3058,B 24.8814,C -2.5138,E1 25.0979,E2 142.0588} C_DIS
LIN {X 35.8999,Y -43.1944,Z 70,A -54.8107,B 24.8806,C -2.5224,E1 25.1054,E2 138.5567} C_DIS
LIN {X 38.7408,Y -40.6668,Z 70,A -51.7682,B 24.8815,C -2.5127,E1 25.1116,E2 135.5495} C_DIS
LIN {X 40.1793,Y -39.2462,Z 70,A -49.7464,B 24.8811,C -2.5167,E1 25.1156,E2 133.5267} C_DIS
LIN {X 42.9785,Y -36.1596,Z 70,A -45.7047,B 24.8805,C -2.5227,E1 25.1231,E2 129.4889} C_DIS
LIN {X 44.8828,Y -33.7653,Z 70,A -41.8604,B 24.8782,C -2.5472,E1 25.1297,E2 125.605} C_DIS
LIN {X 46.9702,Y -30.7957,Z 70,A -38.4862,B 24.8779,C -2.5498,E1 25.135,E2 122.2411} C_DIS
LIN {X 48.9813,Y -27.4845,Z 70,A -34.9648,B 24.8779,C -2.5513,E1 25.14,E2 118.7343} C_DIS
LIN {X 50.3208,Y -24.9475,Z 70,A -31.2779,B 24.8753,C -2.5771,E1 25.1447,E2 115.006} C_DIS
LIN {X 51.7186,Y -21.9016,Z 70,A -27.9155,B 24.8744,C -2.586,E1 25.1484,E2 111.6409} C_DIS
LIN {X 53.3277,Y -17.6302,Z 70,A -23.8813,B 24.8744,C -2.5859,E1 25.1522,E2 107.6296} C_DIS
LIN {X 53.9899,Y -15.4816,Z 70,A -20.9183,B 24.8723,C -2.6083,E1 25.1546,E2 104.6304} C_DIS
LIN {X 54.7862,Y -12.3734,Z 70,A -18.4543,B 24.8731,C -2.6,E1 25.1561,E2 102.2005} C_DIS
LIN {X 55.4601,Y -8.8781,Z 70,A -14.6993,B 24.8717,C -2.6142,E1 25.158,E2 98.4338} C_DIS
LIN {X 55.8508,Y -5.9375,Z 70,A -11.1978,B 24.8697,C -2.6347,E1 25.1592,E2 94.9046} C_DIS
LIN {X 56.1091,Y -2.5166,Z 70,A -8.197,B 24.8697,C -2.6343,E1 25.1597,E2 91.9225} C_DIS
LIN {X 56.1668,Y 0.2,Z 70,A -5.4342,B 24.8689,C -2.6428,E1 25.1597,E2 89.1561} C_DIS
LIN {X 55.9905,Y 4.4293,Z 70,A -0.637,B 24.8664,C -2.6673,E1 25.159,E2 84.3293} C_DIS
LIN {X 55.5762,Y 8.117,Z 70,A 2.6392,B 24.8664,C -2.6673,E1 25.1578,E2 81.0724} C_DIS
LIN {X 55.1477,Y 10.6439,Z 70,A 5.3354,B 24.8654,C -2.6773,E1 25.1565,E2 78.3686} C_DIS
LIN {X 54.4955,Y 13.5963,Z 70,A 8.3622,B 24.8646,C -2.6853,E1 25.1545,E2 75.3404} C_DIS
LIN {X 53.8757,Y 15.8736,Z 70,A 10.5349,B 24.8644,C -2.6871,E1 25.1529,E2 73.1757} C_DIS
LIN {X 52.9179,Y 18.823,Z 70,A 13.7862,B 24.8633,C -2.6984,E1 25.15,E2 69.9162} C_DIS
LIN {X 51.8421,Y 21.6098,Z 70,A 16.7159,B 24.8626,C -2.7044,E1 25.147,E2 66.9884} C_DIS
LIN {X 51.0557,Y 23.406,Z 70,A 19.1705,B 24.861,C -2.7202,E1 25.1441,E2 64.5098} C_DIS
LIN {X 49.1752,Y 27.1373,Z 70,A 23.6062,B 24.8595,C -2.7355,E1 25.1383,E2 60.0612} C_DIS
LIN {X 47.3732,Y 30.1724,Z 70,A 26.7801,B 24.8595,C -2.7353,E1 25.1337,E2 56.904} C_DIS
LIN {X 45.4429,Y 33.0082,Z 70,A 30.6803,B 24.8577,C -2.7528,E1 25.1274,E2 52.9815} C_DIS
LIN {X 43.4292,Y 35.6169,Z 70,A 33.6442,B 24.8577,C -2.7518,E1 25.1222,E2 50.0336} C_DIS
LIN {X 41.4927,Y 37.8542,Z 70,A 36.3135,B 24.8579,C -2.7509,E1 25.1173,E2 47.3784} C_DIS
LIN {X 40.2651,Y 39.1579,Z 70,A 38.7349,B 24.8561,C -2.7677,E1 25.1125,E2 44.9276} C_DIS
LIN {X 37.7454,Y 41.5925,Z 70,A 41.9199,B 24.8562,C -2.7665,E1 25.1061,E2 41.7586} C_DIS
LIN {X 35.4125,Y 43.5949,Z 70,A 45.3599,B 24.855,C -2.7788,E1 25.0987,E2 38.3025} C_DIS
LIN {X 32.7378,Y 45.6378,Z 70,A 49.1179,B 24.8536,C -2.7916,E1 25.0901,E2 34.5275} C_DIS
LIN {X 29.6916,Y 47.6757,Z 70,A 52.0111,B 24.8549,C -2.7795,E1 25.0834,E2 31.6725} C_DIS
LIN {X 27.202,Y 49.1391,Z 70,A 55.5159,B 24.8532,C -2.7953,E1 25.0749,E2 28.1408} C_DIS
LIN {X 22.8159,Y 51.3232,Z 70,A 60.5747,B 24.8525,C -2.8023,E1 25.0621,E2 23.0782} C_DIS
LIN {X 19.4788,Y 52.68,Z 70,A 64.2815,B 24.852,C -2.8064,E1 25.0524,E2 19.3697} C_DIS
LIN {X 15.2101,Y 54.0668,Z 70,A 68.3294,B 24.8528,C -2.799,E1 25.0417,E2 15.3467} C_DIS
LIN {X 12.5261,Y 54.751,Z 70,A 70.9939,B 24.853,C -2.7973,E1 25.0345,E2 12.69} C_DIS
LIN {X 10.4767,Y 55.1798,Z 70,A 73.2347,B 24.8527,C -2.8003,E1 25.0283,E2 10.4448} C_DIS
LIN {X 8.1113,Y 55.5771,Z 70,A 75.6281,B 24.8527,C -2.8,E1 25.0217,E2 8.0544} C_DIS
LIN {X 5.8868,Y 55.8561,Z 70,A 77.8801,B 24.8527,C -2.7997,E1 25.0155,E2 5.8048} C_DIS
LIN {X 3.6015,Y 56.0501,Z 70,A 80.3885,B 24.8524,C -2.8031,E1 25.0085,E2 3.2896} C_DIS
LIN {X 1.173,Y 56.1534,Z 70,A 82.6468,B 24.8529,C -2.7986,E1 25.0022,E2 1.0426} C_DIS
LIN {X -1.7021,Y 56.1396,Z 70,A 86.0437,B 24.852,C -2.8068,E1 24.9927,E2 -2.374} C_DIS
LIN {X -4.7622,Y 55.9635,Z 70,A 88.9173,B 24.8527,C -2.8006,E1 24.9847,E2 -5.2341} C_DIS
LIN {X -6.9618,Y 55.7324,Z 70,A 91.4628,B 24.8522,C -2.8048,E1 24.9776,E2 -7.7913} C_DIS
LIN {X -10.6785,Y 55.141,Z 70,A 94.7694,B 24.8536,C -2.792,E1 24.9686,E2 -11.0708} C_DIS
LIN {X -12.5666,Y 54.7416,Z 70,A 96.8936,B 24.8534,C -2.7932,E1 24.9628,E2 -13.2004} C_DIS
LIN {X -14.8631,Y 54.1636,Z 70,A 99.3128,B 24.8537,C -2.7909,E1 24.9563,E2 -15.6177} C_DIS
LIN {X -17.0677,Y 53.5096,Z 70,A 101.9025,B 24.8535,C -2.7927,E1 24.9493,E2 -18.2163} C_DIS
LIN {X -19.8913,Y 52.5252,Z 70,A 104.6064,B 24.8546,C -2.7826,E1 24.9423,E2 -20.9015} C_DIS
LIN {X -22.2843,Y 51.5558,Z 70,A 107.4815,B 24.8545,C -2.7833,E1 24.9348,E2 -23.7848} C_DIS
LIN {X -24.684,Y 50.4514,Z 70,A 110.1514,B 24.855,C -2.7787,E1 24.9281,E2 -26.4505} C_DIS
LIN {X -27.0913,Y 49.2003,Z 70,A 112.924,B 24.8554,C -2.7742,E1 24.9213,E2 -29.2202} C_DIS
LIN {X -30.2596,Y 47.3168,Z 70,A 117.4904,B 24.8547,C -2.7816,E1 24.9104,E2 -33.8186} C_DIS
LIN {X -32.8585,Y 45.5517,Z 70,A 120.4546,B 24.8558,C -2.771,E1 24.9037,E2 -36.7677} C_DIS
LIN {X -36.7933,Y 42.4364,Z 70,A 124.9197,B 24.8581,C -2.7486,E1 24.8941,E2 -41.1963} C_DIS
LIN {X -39.6173,Y 39.8129,Z 70,A 128.9784,B 24.8588,C -2.7417,E1 24.8859,E2 -45.2551} C_DIS
LIN {X -41.1951,Y 38.1785,Z 70,A 131.6426,B 24.8588,C -2.7419,E1 24.8808,E2 -47.9316} C_DIS
LIN {X -43.8885,Y 35.049,Z 70,A 135.2307,B 24.861,C -2.7207,E1 24.8744,E2 -51.4855} C_DIS
LIN {X -45.3926,Y 33.077,Z 70,A 138.6657,B 24.8601,C -2.7292,E1 24.8686,E2 -54.9573} C_DIS
LIN {X -47.386,Y 30.1517,Z 70,A 142.246,B 24.8612,C -2.7188,E1 24.8632,E2 -58.5307} C_DIS
LIN {X -49.6077,Y 26.3376,Z 70,A 146.1276,B 24.8635,C -2.6957,E1 24.8579,E2 -62.3774} C_DIS
LIN {X -50.4427,Y 24.6998,Z 70,A 148.3114,B 24.8635,C -2.6953,E1 24.8552,E2 -64.572} C_DIS
LIN {X -51.8803,Y 21.5196,Z 70,A 152.1328,B 24.8642,C -2.689,E1 24.8509,E2 -68.3995} C_DIS
LIN {X -53.3851,Y 17.4532,Z 70,A 156.3071,B 24.866,C -2.6715,E1 24.8471,E2 -72.5556} C_DIS
LIN {X -54.0402,Y 15.3041,Z 70,A 158.9314,B 24.8661,C -2.6699,E1 24.8451,E2 -75.1912} C_DIS
LIN {X -54.7701,Y 12.4406,Z 70,A 162.1172,B 24.8668,C -2.6633,E1 24.843,E2 -78.38} C_DIS
LIN {X -55.3987,Y 9.2491,Z 70,A 165.0301,B 24.8685,C -2.6462,E1 24.8416,E2 -81.2694} C_DIS
LIN {X -55.8623,Y 5.8274,Z 70,A 168.8128,B 24.8692,C -2.6394,E1 24.8404,E2 -85.0584} C_DIS
LIN {X -56.089,Y 2.9338,Z 70,A 172.1118,B 24.8696,C -2.6356,E1 24.8398,E2 -88.3681} C_DIS
LIN {X -56.0941,Y -2.842,Z 70,A 178.03,B 24.8714,C -2.6175,E1 24.8402,E2 -94.2786} C_DIS
LIN {X -55.7009,Y -7.2084,Z 70,A -177.7197,B 24.8731,C -2.5999,E1 24.8415,E2 -98.5124} C_DIS
LIN {X -54.9159,Y -11.7831,Z 70,A -172.6139,B 24.8739,C -2.5916,E1 24.8443,E2 -103.6285} C_DIS
LIN {X -53.6944,Y -16.4771,Z 70,A -168.2447,B 24.8763,C -2.5672,E1 24.8475,E2 -107.9647} C_DIS
LIN {X -52.5538,Y -19.8155,Z 70,A -164.6759,B 24.8773,C -2.5563,E1 24.8509,E2 -111.5276} C_DIS
LIN {X -51.8014,Y -21.7067,Z 70,A -162.7259,B 24.8781,C -2.5483,E1 24.8529,E2 -113.4694} C_DIS
LIN {X -51.143,Y -23.2158,Z 70,A -160.2509,B 24.8773,C -2.5571,E1 24.8559,E2 -115.9789} C_DIS
LIN {X -49.4285,Y -26.6719,Z 70,A -155.8398,B 24.8775,C -2.5547,E1 24.8617,E2 -120.4077} C_DIS
LIN {X -47.5922,Y -29.8253,Z 70,A -152.1044,B 24.8784,C -2.5454,E1 24.8672,E2 -124.1399} C_DIS
LIN {X -45.5532,Y -32.8564,Z 70,A -149.4386,B 24.881,C -2.5178,E1 24.8714,E2 -126.753} C_DIS
LIN {X -43.8276,Y -35.1253,Z 70,A -146.8776,B 24.8822,C -2.505,E1 24.8758,E2 -129.2955} C_DIS
LIN {X -41.9889,Y -37.3033,Z 70,A -143.465,B 24.882,C -2.5073,E1 24.882,E2 -132.7289} C_DIS
LIN {X -39.7544,Y -39.6763,Z 70,A -139.9421,B 24.8823,C -2.5037,E1 24.8889,E2 -136.2585} C_DIS
LIN {X -37.0379,Y -42.2228,Z 70,A -136.4207,B 24.8835,C -2.4914,E1 24.8962,E2 -139.7646} C_DIS
LIN {X -34.8605,Y -44.0376,Z 70,A -133.627,B 24.8841,C -2.4844,E1 24.9022,E2 -142.5522} C_DIS
LIN {X -32.8352,Y -45.5684,Z 70,A -130.556,B 24.8837,C -2.4887,E1 24.9092,E2 -145.6443} C_DIS
LIN {X -29.7649,Y -47.6299,Z 70,A -126.9768,B 24.8846,C -2.4795,E1 24.9175,E2 -149.213} C_DIS
LIN {X -26.5045,Y -49.5194,Z 70,A -123.1183,B 24.8851,C -2.4746,E1 24.9269,E2 -153.0709} C_DIS
LIN {X -23.1091,Y -51.1911,Z 70,A -118.879,B 24.8848,C -2.4773,E1 24.9377,E2 -157.3274} C_DIS
LIN {X -18.9542,Y -52.8714,Z 70,A -114.72,B 24.8859,C -2.4652,E1 24.9485,E2 -161.4665} C_DIS
LIN {X -15.7028,Y -53.9253,Z 70,A -111.5186,B 24.8867,C -2.4573,E1 24.957,E2 -164.6547} C_DIS
LIN {X -13.3927,Y -54.5453,Z 70,A -108.837,B 24.8864,C -2.4606,E1 24.9643,E2 -167.3479} C_DIS
LIN {X -10.3799,Y -55.1971,Z 70,A -106.1613,B 24.8873,C -2.4503,E1 24.9715,E2 -170.0022} C_DIS
LIN {X -8.7432,Y -55.481,Z 70,A -104.0069,B 24.8865,C -2.4587,E1 24.9775,E2 -172.1786} C_DIS
LIN {X -6.2658,Y -55.8153,Z 70,A -101.7421,B 24.8871,C -2.4527,E1 24.9838,E2 -174.4308} C_DIS
LIN {X -3.9063,Y -56.0296,Z 70,A -99.0808,B 24.8867,C -2.4575,E1 24.9912,E2 -177.1045} C_DIS
LIN {X -0.0641,Y -56.1661,Z 70,A -95.1164,B 24.8865,C -2.4589,E1 25.0023,E2 -181.0728} C_DIS
LIN {X -0.0641,Y -56.1661,Z 70,A -95.1164,B 24.8865,C -2.4589,E1 25.0023,E2 -181.0728} C_DIS
Enddeposition()
LIN {X 0.2988,Y -55.2114,Z 70,A -95.1723,B 24.8858,C -2.4669,E1 25.0022,E2 -181.0359} C_DIS
Startdeposition()
$VEL.CP = VEL_PRINT
LIN {X -1.903,Y -55.1808,Z 70,A -98.482,B 24.8876,C -2.4467,E1 24.9928,E2 -177.678} C_DIS
LIN {X -4.1794,Y -55.0559,Z 70,A -100.6714,B 24.8873,C -2.45,E1 24.9867,E2 -175.4956} C_DIS
LIN {X -6.3915,Y -54.8428,Z 70,A -103.1582,B 24.8876,C -2.4468,E1 24.9798,E2 -172.9998} C_DIS
LIN {X -8.9733,Y -54.4801,Z 70,A -105.9059,B 24.8876,C -2.4468,E1 24.9722,E2 -170.2495} C_DIS
LIN {X -11.8884,Y -53.9182,Z 70,A -109.1316,B 24.8878,C -2.4454,E1 24.9634,E2 -167.0166} C_DIS
LIN {X -14.9256,Y -53.1586,Z 70,A -112.5166,B 24.8878,C -2.4448,E1 24.9542,E2 -163.6253} C_DIS
LIN {X -18.6384,Y -51.9739,Z 70,A -116.2398,B 24.887,C -2.4538,E1 24.9444,E2 -159.9164} C_DIS
LIN {X -20.6571,Y -51.2045,Z 70,A -118.2851,B 24.8865,C -2.4594,E1 24.9391,E2 -157.8802} C_DIS
LIN {X -22.823,Y -50.2765,Z 70,A -120.9581,B 24.8866,C -2.458,E1 24.9323,E2 -155.1973} C_DIS
LIN {X -25.7763,Y -48.828,Z 70,A -124.9501,B 24.8872,C -2.452,E1 24.9223,E2 -151.1803} C_DIS
LIN {X -29.0654,Y -46.9451,Z 70,A -128.175,B 24.8855,C -2.4699,E1 24.9146,E2 -147.9882} C_DIS
LIN {X -31.9463,Y -45.0338,Z 70,A -131.3893,B 24.8844,C -2.482,E1 24.9072,E2 -144.7922} C_DIS
LIN {X -33.4039,Y -43.9643,Z 70,A -133.8455,B 24.885,C -2.4752,E1 24.9017,E2 -142.311} C_DIS
LIN {X -35.544,Y -42.2531,Z 70,A -136.7067,B 24.8845,C -2.4801,E1 24.8955,E2 -139.4506} C_DIS
LIN {X -37.6366,Y -40.3997,Z 70,A -140.113,B 24.8848,C -2.4774,E1 24.8884,E2 -136.024} C_DIS
LIN {X -40.0266,Y -38.0334,Z 70,A -143.1416,B 24.8834,C -2.4924,E1 24.8826,E2 -133.0181} C_DIS
LIN {X -42.2928,Y -35.4962,Z 70,A -146.5931,B 24.8825,C -2.5015,E1 24.8763,E2 -129.573} C_DIS
LIN {X -43.9717,Y -33.394,Z 70,A -149.5285,B 24.8821,C -2.5057,E1 24.8712,E2 -126.6337} C_DIS
LIN {X -46.2869,Y -30.1023,Z 70,A -153.545,B 24.8809,C -2.5187,E1 24.8649,E2 -122.6282} C_DIS
LIN {X -47.8622,Y -27.5281,Z 70,A -156.9933,B 24.8806,C -2.5217,E1 24.86,E2 -119.1693} C_DIS
LIN {X -48.9888,Y -25.471,Z 70,A -159.3551,B 24.8799,C -2.5294,E1 24.8569,E2 -116.8133} C_DIS
LIN {X -50.1272,Y -23.1491,Z 70,A -161.9446,B 24.8791,C -2.5383,E1 24.8538,E2 -114.231} C_DIS
LIN {X -51.2556,Y -20.5315,Z 70,A -164.9467,B 24.8783,C -2.5459,E1 24.8506,E2 -111.2305} C_DIS
LIN {X -52.3099,Y -17.6711,Z 70,A -167.8651,B 24.8771,C -2.559,E1 24.8478,E2 -108.3268} C_DIS
LIN {X -53.0768,Y -15.2136,Z 70,A -171.0027,B 24.8771,C -2.5595,E1 24.8453,E2 -105.1723} C_DIS
LIN {X -53.8063,Y -12.3882,Z 70,A -173.809,B 24.8758,C -2.5721,E1 24.8435,E2 -102.3797} C_DIS
LIN {X -54.4253,Y -9.301,Z 70,A -177.2206,B 24.875,C -2.5798,E1 24.8417,E2 -98.9665} C_DIS
LIN {X -54.82,Y -6.5862,Z 70,A 179.6628,B 24.8746,C -2.5845,E1 24.8406,E2 -95.8423} C_DIS
LIN {X -55.1236,Y -3.1607,Z 70,A 176.3677,B 24.8731,C -2.5999,E1 24.8399,E2 -92.5641} C_DIS
LIN {X -55.2099,Y 0.7293,Z 70,A 171.8253,B 24.8726,C -2.6048,E1 24.8399,E2 -88.0061} C_DIS
LIN {X -55.098,Y 3.5803,Z 70,A 168.7182,B 24.8719,C -2.6119,E1 24.8404,E2 -84.8973} C_DIS
LIN {X -54.504,Y 8.8305,Z 70,A 164.1255,B 24.8688,C -2.6429,E1 24.842,E2 -80.3514} C_DIS
LIN {X -54.0603,Y 11.229,Z 70,A 161.2214,B 24.8686,C -2.645,E1 24.8436,E2 -77.4352} C_DIS
LIN {X -53.378,Y 14.1223,Z 70,A 158.4118,B 24.8672,C -2.6589,E1 24.8455,E2 -74.6423} C_DIS
LIN {X -52.7382,Y 16.3485,Z 70,A 155.8033,B 24.8668,C -2.6631,E1 24.8475,E2 -72.0288} C_DIS
LIN {X -51.4011,Y 20.1622,Z 70,A 151.5459,B 24.8656,C -2.6748,E1 24.8516,E2 -67.7753} C_DIS
LIN {X -50.0385,Y 23.3394,Z 70,A 147.7434,B 24.8649,C -2.682,E1 24.8559,E2 -63.9692} C_DIS
LIN {X -48.8793,Y 25.6788,Z 70,A 145.3136,B 24.8637,C -2.6943,E1 24.859,E2 -61.5557} C_DIS
LIN {X -47.8219,Y 27.5976,Z 70,A 142.2773,B 24.8642,C -2.6887,E1 24.8632,E2 -58.4903} C_DIS
LIN {X -46.1335,Y 30.3364,Z 70,A 139.5187,B 24.8624,C -2.7071,E1 24.8674,E2 -55.7615} C_DIS
LIN {X -43.6563,Y 33.8044,Z 70,A 135.4222,B 24.8606,C -2.724,E1 24.8741,E2 -51.6858} C_DIS
LIN {X -41.5676,Y 36.3417,Z 70,A 131.2008,B 24.8611,C -2.7197,E1 24.8817,E2 -47.4345} C_DIS
LIN {X -39.7039,Y 38.3692,Z 70,A 127.6754,B 24.8615,C -2.7159,E1 24.8886,E2 -43.8849} C_DIS
LIN {X -37.1038,Y 40.89,Z 70,A 124.9943,B 24.8588,C -2.7418,E1 24.894,E2 -41.2549} C_DIS
LIN {X -33.1708,Y 44.1393,Z 70,A 119.9138,B 24.8573,C -2.7566,E1 24.905,E2 -36.1907} C_DIS
LIN {X -30.6647,Y 45.9161,Z 70,A 116.262,B 24.8574,C -2.7551,E1 24.9134,E2 -32.5229} C_DIS
LIN {X -27.5747,Y 47.8354,Z 70,A 112.9488,B 24.8559,C -2.7697,E1 24.9213,E2 -29.2342} C_DIS
LIN {X -26.0493,Y 48.6828,Z 70,A 110.7263,B 24.8563,C -2.7657,E1 24.9268,E2 -26.996} C_DIS
LIN {X -22.8614,Y 50.2592,Z 70,A 107.4504,B 24.855,C -2.7785,E1 24.935,E2 -23.7421} C_DIS
LIN {X -21.2104,Y 50.9781,Z 70,A 105.2432,B 24.8553,C -2.7752,E1 24.9407,E2 -21.5222} C_DIS
LIN {X -18.5697,Y 51.9984,Z 70,A 102.3961,B 24.8548,C -2.7806,E1 24.9481,E2 -18.6818} C_DIS
LIN {X -14.7607,Y 53.2053,Z 70,A 97.2831,B 24.8561,C -2.7682,E1 24.9619,E2 -13.531} C_DIS
LIN {X -10.4819,Y 54.2099,Z 70,A 93.6799,B 24.8539,C -2.789,E1 24.9716,E2 -9.9728} C_DIS
LIN {X -8.0919,Y 54.6176,Z 70,A 91.1719,B 24.8537,C -2.7909,E1 24.9785,E2 -7.4671} C_DIS
LIN {X -5.4072,Y 54.949,Z 70,A 88.5557,B 24.8532,C -2.7959,E1 24.9857,E2 -4.8611} C_DIS
LIN {X -3.8099,Y 55.0825,Z 70,A 86.1404,B 24.8545,C -2.7829,E1 24.9926,E2 -2.414} C_DIS
LIN {X 1.0567,Y 55.2039,Z 70,A 81.8348,B 24.853,C -2.7978,E1 25.0045,E2 1.8564} C_DIS
LIN {X 2.6877,Y 55.1486,Z 70,A 79.6195,B 24.854,C -2.7881,E1 25.0107,E2 4.0938} C_DIS
LIN {X 6.1123,Y 54.8755,Z 70,A 76.1692,B 24.8538,C -2.7899,E1 25.0203,E2 7.5378} C_DIS
LIN {X 9.5145,Y 54.3874,Z 70,A 72.8861,B 24.8533,C -2.7942,E1 25.0293,E2 10.8074} C_DIS
LIN {X 11.7201,Y 53.9558,Z 70,A 70.1152,B 24.8543,C -2.7848,E1 25.0369,E2 13.5973} C_DIS
LIN {X 15.4495,Y 53.0091,Z 70,A 66.6577,B 24.8535,C -2.7926,E1 25.0462,E2 17.0308} C_DIS
LIN {X 17.1792,Y 52.4737,Z 70,A 64.6627,B 24.8539,C -2.7889,E1 25.0515,E2 19.0309} C_DIS
LIN {X 19.5594,Y 51.6335,Z 70,A 61.9073,B 24.8544,C -2.7839,E1 25.0588,E2 21.7925} C_DIS
LIN {X 22.8552,Y 50.262,Z 70,A 57.9303,B 24.8554,C -2.7745,E1 25.069,E2 25.7821} C_DIS
LIN {X 25.0463,Y 49.2065,Z 70,A 55.6091,B 24.8554,C -2.7754,E1 25.0748,E2 28.0948} C_DIS
LIN {X 27.6533,Y 47.7896,Z 70,A 52.1012,B 24.8566,C -2.7626,E1 25.0833,E2 31.6227} C_DIS
LIN {X 30.8582,Y 45.7862,Z 70,A 48.7135,B 24.8562,C -2.7673,E1 25.0912,E2 34.9882} C_DIS
LIN {X 33.1227,Y 44.1755,Z 70,A 45.8673,B 24.8566,C -2.7632,E1 25.0976,E2 37.8341} C_DIS
LIN {X 36.1675,Y 41.7198,Z 70,A 41.9611,B 24.857,C -2.7588,E1 25.106,E2 41.7357} C_DIS
LIN {X 37.9737,Y 40.0827,Z 70,A 39.1592,B 24.8582,C -2.7481,E1 25.1118,E2 44.5515} C_DIS
LIN {X 40.8161,Y 37.1843,Z 70,A 35.1559,B 24.8586,C -2.7435,E1 25.1195,E2 48.5485} C_DIS
LIN {X 42.5804,Y 35.1501,Z 70,A 32.3476,B 24.8593,C -2.7368,E1 25.1246,E2 51.3598} C_DIS
LIN {X 44.2964,Y 32.9618,Z 70,A 28.6453,B 24.8618,C -2.7127,E1 25.1309,E2 55.1014} C_DIS
LIN {X 46.5775,Y 29.6507,Z 70,A 25.3119,B 24.8611,C -2.72,E1 25.1359,E2 58.401} C_DIS
LIN {X 48.1994,Y 26.9333,Z 70,A 21.3739,B 24.8634,C -2.6974,E1 25.1414,E2 62.3721} C_DIS
LIN {X 50.616,Y 22.0591,Z 70,A 17.0451,B 24.862,C -2.7103,E1 25.1466,E2 66.6471} C_DIS
LIN {X 51.594,Y 19.6636,Z 70,A 13.632,B 24.8644,C -2.6868,E1 25.1502,E2 70.097} C_DIS
LIN {X 52.5165,Y 17.0471,Z 70,A 10.84,B 24.8651,C -2.6802,E1 25.1527,E2 72.8886} C_DIS
LIN {X 53.3562,Y 14.2036,Z 70,A 8.0886,B 24.8653,C -2.6782,E1 25.1547,E2 75.6291} C_DIS
LIN {X 53.8175,Y 12.3398,Z 70,A 5.92,B 24.8663,C -2.6683,E1 25.1561,E2 77.8085} C_DIS
LIN {X 54.3697,Y 9.6199,Z 70,A 3.1658,B 24.8669,C -2.6623,E1 25.1576,E2 80.5609} C_DIS
LIN {X 54.7455,Y 7.1784,Z 70,A 0.5914,B 24.8677,C -2.6541,E1 25.1586,E2 83.1395} C_DIS
LIN {X 55.0499,Y 4.2558,Z 70,A -2.9168,B 24.8697,C -2.6345,E1 25.1595,E2 86.6733} C_DIS
LIN {X 55.1971,Y 1.3975,Z 70,A -5.4242,B 24.8696,C -2.6353,E1 25.1598,E2 89.1638} C_DIS
LIN {X 55.1949,Y -1.4693,Z 70,A -8.4218,B 24.8706,C -2.6254,E1 25.1597,E2 92.1669} C_DIS
LIN {X 55.0657,Y -4.0575,Z 70,A -11.484,B 24.8722,C -2.6087,E1 25.1591,E2 95.2504} C_DIS
LIN {X 54.7193,Y -7.3805,Z 70,A -14.5516,B 24.8724,C -2.6066,E1 25.1581,E2 98.305} C_DIS
LIN {X 54.1822,Y -10.6238,Z 70,A -17.8794,B 24.8733,C -2.5977,E1 25.1565,E2 101.6342} C_DIS
LIN {X 53.6852,Y -12.9044,Z 70,A -20.6417,B 24.8748,C -2.5826,E1 25.1547,E2 104.4161} C_DIS
LIN {X 52.5698,Y -16.8826,Z 70,A -24.0643,B 24.8742,C -2.5885,E1 25.1521,E2 107.8053} C_DIS
LIN {X 51.6335,Y -19.5594,Z 70,A -28.1194,B 24.8774,C -2.5551,E1 25.1482,E2 111.9168} C_DIS
LIN {X 50.1001,Y -23.2072,Z 70,A -32.4224,B 24.879,C -2.5386,E1 25.1432,E2 116.2353} C_DIS
LIN {X 48.358,Y -26.6493,Z 70,A -35.9797,B 24.8792,C -2.5367,E1 25.1385,E2 119.7783} C_DIS
LIN {X 46.5264,Y -29.7304,Z 70,A -39.0845,B 24.8789,C -2.5397,E1 25.134,E2 122.8604} C_DIS
LIN {X 45.4709,Y -31.3215,Z 70,A -41.3549,B 24.88,C -2.528,E1 25.1304,E2 125.1473} C_DIS
LIN {X 43.5736,Y -33.9116,Z 70,A -44.2264,B 24.88,C -2.5291,E1 25.1257,E2 128.0024} C_DIS
LIN {X 42.3497,Y -35.4277,Z 70,A -46.5737,B 24.8811,C -2.5168,E1 25.1215,E2 130.3678} C_DIS
LIN {X 40.0185,Y -38.0394,Z 70,A -50.1459,B 24.8818,C -2.5091,E1 25.1148,E2 133.9425} C_DIS
LIN {X 37.96,Y -40.0946,Z 70,A -53.4017,B 24.883,C -2.4969,E1 25.1082,E2 137.2135} C_DIS
LIN {X 36.1216,Y -41.7599,Z 70,A -55.7747,B 24.8831,C -2.4954,E1 25.1032,E2 139.5808} C_DIS
LIN {X 33.4044,Y -43.9628,Z 70,A -59.5041,B 24.884,C -2.4856,E1 25.095,E2 143.3196} C_DIS
LIN {X 30.7657,Y -45.8488,Z 70,A -62.5133,B 24.884,C -2.4863,E1 25.0882,E2 146.3166} C_DIS
LIN {X 29.1392,Y -46.899,Z 70,A -64.4325,B 24.8841,C -2.4844,E1 25.0837,E2 148.2342} C_DIS
LIN {X 27.1269,Y -48.0913,Z 70,A -67.0751,B 24.885,C -2.4756,E1 25.0773,E2 150.8896} C_DIS
LIN {X 23.1168,Y -50.1422,Z 70,A -71.2077,B 24.8846,C -2.4793,E1 25.067,E2 155.0023} C_DIS
LIN {X 20.8202,Y -51.1381,Z 70,A -74.8336,B 24.8869,C -2.4545,E1 25.0575,E2 158.6784} C_DIS
LIN {X 16.204,Y -52.783,Z 70,A -79.9775,B 24.8876,C -2.4472,E1 25.0439,E2 163.8299} C_DIS
LIN {X 11.7413,Y -53.9512,Z 70,A -84.1648,B 24.8869,C -2.4545,E1 25.0326,E2 167.9937} C_DIS
LIN {X 9.1327,Y -54.4535,Z 70,A -86.9925,B 24.8873,C -2.4509,E1 25.0248,E2 170.8268} C_DIS
LIN {X 4.5211,Y -55.0287,Z 70,A -91.4023,B 24.8868,C -2.4561,E1 25.0126,E2 175.2209} C_DIS
LIN {X 2.5323,Y -55.1561,Z 70,A -93.8108,B 24.8875,C -2.4487,E1 25.0059,E2 177.6462} C_DIS
LIN {X 0.2988,Y -55.2114,Z 70,A -95.1716,B 24.8858,C -2.4666,E1 25.0022,E2 178.9641} C_DIS
Enddeposition()
LIN {X 0.2988,Y -55.2114,Z 70,A -95.1716,B 24.8858,C -2.4666,E1 25.0022,E2 178.9641} C_DIS
Startdeposition()
$VEL.CP = VEL_PRINT
LIN {X 1.499,Y -54.2421,Z 70,A -93.6743,B 24.8838,C -2.4878,E1 25.0065,E2 177.4168} C_DIS
LIN {X 4.16,Y -54.1031,Z 70,A -90.8787,B 24.8838,C -2.4886,E1 25.0143,E2 174.6204} C_DIS
LIN {X 5.8625,Y -53.9454,Z 70,A -88.7779,B 24.8831,C -2.4955,E1 25.0202,E2 172.5048} C_DIS
LIN {X 8.9989,Y -53.5112,Z 70,A -85.6697,B 24.8833,C -2.4932,E1 25.0287,E2 169.405} C_DIS
LIN {X 11.4415,Y -53.0428,Z 70,A -82.4977,B 24.8821,C -2.5064,E1 25.0375,E2 166.2057} C_DIS
LIN {X 15.2548,Y -52.0745,Z 70,A -78.9176,B 24.8828,C -2.4991,E1 25.0471,E2 162.6485} C_DIS
LIN {X 17.6801,Y -51.3024,Z 70,A -76.1745,B 24.8824,C -2.5035,E1 25.0543,E2 159.9003} C_DIS
LIN {X 19.6632,Y -50.5749,Z 70,A -73.8427,B 24.8819,C -2.5086,E1 25.0604,E2 157.5615} C_DIS
LIN {X 22.7481,Y -49.2644,Z 70,A -70.5646,B 24.8819,C -2.5084,E1 25.0688,E2 154.2918} C_DIS
LIN {X 25.5419,Y -47.8761,Z 70,A -67.1669,B 24.8812,C -2.516,E1 25.0773,E2 150.8855} C_DIS
LIN {X 28.0369,Y -46.4584,Z 70,A -64.5481,B 24.8815,C -2.5128,E1 25.0836,E2 148.2822} C_DIS
LIN {X 29.3971,Y -45.6095,Z 70,A -62.7724,B 24.881,C -2.5177,E1 25.0878,E2 146.5006} C_DIS
LIN {X 31.3234,Y -44.3084,Z 70,A -59.8939,B 24.8797,C -2.5315,E1 25.0944,E2 143.5992} C_DIS
LIN {X 34.2755,Y -42.0671,Z 70,A -56.1433,B 24.8792,C -2.5363,E1 25.1027,E2 139.8511} C_DIS
LIN {X 36.3508,Y -40.2876,Z 70,A -53.2565,B 24.8786,C -2.5428,E1 25.1087,E2 136.9603} C_DIS
LIN {X 38.598,Y -38.1395,Z 70,A -49.69,B 24.8773,C -2.5567,E1 25.1159,E2 133.3759} C_DIS
LIN {X 40.8229,Y -35.7481,Z 70,A -46.5787,B 24.8772,C -2.558,E1 25.1217,E2 130.2754} C_DIS
LIN {X 42.5438,Y -33.6817,Z 70,A -43.8776,B 24.8767,C -2.5624,E1 25.1264,E2 127.5765} C_DIS
LIN {X 43.9234,Y -31.8619,Z 70,A -41.3133,B 24.8758,C -2.5721,E1 25.1307,E2 125.0014} C_DIS
LIN {X 45.2261,Y -29.9835,Z 70,A -38.6078,B 24.8745,C -2.5852,E1 25.1349,E2 122.2785} C_DIS
LIN {X 47.5333,Y -26.1748,Z 70,A -34.2295,B 24.8739,C -2.5913,E1 25.1411,E2 117.9082} C_DIS
LIN {X 49.0032,Y -23.3059,Z 70,A -30.8242,B 24.873,C -2.6013,E1 25.1453,E2 114.4974} C_DIS
LIN {X 49.9849,Y -21.1174,Z 70,A -27.5779,B 24.8706,C -2.6248,E1 25.1489,E2 111.2135} C_DIS
LIN {X 51.4871,Y -17.1333,Z 70,A -23.9334,B 24.8712,C -2.6195,E1 25.1522,E2 107.6019} C_DIS
LIN {X 52.2219,Y -14.7414,Z 70,A -21.3015,B 24.8704,C -2.6274,E1 25.1543,E2 104.9663} C_DIS
LIN {X 52.7474,Y -12.7342,Z 70,A -18.9784,B 24.8694,C -2.6372,E1 25.1559,E2 102.6336} C_DIS
LIN {X 53.4141,Y -9.5587,Z 70,A -15.6748,B 24.8686,C -2.6452,E1 25.1576,E2 99.3303} C_DIS
LIN {X 53.8151,Y -6.9545,Z 70,A -13.2989,B 24.8686,C -2.645,E1 25.1586,E2 96.9689} C_DIS
LIN {X 54.0388,Y -4.9234,Z 70,A -10.7384,B 24.8671,C -2.6607,E1 25.1593,E2 94.3864} C_DIS
LIN {X 54.2146,Y -2.2829,Z 70,A -8.1251,B 24.8666,C -2.6655,E1 25.1597,E2 91.7772} C_DIS
LIN {X 54.2638,Y 0.2119,Z 70,A -5.3483,B 24.8654,C -2.677,E1 25.1597,E2 88.9899} C_DIS
LIN {X 54.1819,Y 2.9579,Z 70,A -2.6626,B 24.865,C -2.6813,E1 25.1594,E2 86.3098} C_DIS
LIN {X 53.9978,Y 5.3619,Z 70,A -0.0545,B 24.864,C -2.6907,E1 25.1588,E2 83.6952} C_DIS
LIN {X 53.7113,Y 7.7157,Z 70,A 2.5607,B 24.863,C -2.7009,E1 25.1578,E2 81.0711} C_DIS
LIN {X 53.2284,Y 10.5474,Z 70,A 5.1524,B 24.863,C -2.7004,E1 25.1565,E2 78.4957} C_DIS
LIN {X 52.7872,Y 12.5703,Z 70,A 7.4766,B 24.8621,C -2.7101,E1 25.1551,E2 76.1622} C_DIS
LIN {X 52.0611,Y 15.3001,Z 70,A 11.0375,B 24.8599,C -2.7317,E1 25.1524,E2 72.5706} C_DIS
LIN {X 50.6211,Y 19.5457,Z 70,A 15.3232,B 24.8595,C -2.7356,E1 25.1484,E2 68.2998} C_DIS
LIN {X 49.5935,Y 22.0228,Z 70,A 18.1517,B 24.8586,C -2.7435,E1 25.1453,E2 65.4681} C_DIS
LIN {X 48.6513,Y 24.0308,Z 70,A 21.3213,B 24.8561,C -2.7679,E1 25.1413,E2 62.2575} C_DIS
LIN {X 46.4441,Y 28.0606,Z 70,A 25.2482,B 24.8569,C -2.7606,E1 25.1359,E2 58.3683} C_DIS
LIN {X 45.5108,Y 29.5513,Z 70,A 27.4156,B 24.8557,C -2.772,E1 25.1326,E2 56.1848} C_DIS
LIN {X 43.729,Y 32.1281,Z 70,A 30.4397,B 24.8555,C -2.774,E1 25.1277,E2 53.1706} C_DIS
LIN {X 42.0438,Y 34.3042,Z 70,A 33.3212,B 24.8548,C -2.7803,E1 25.1227,E2 50.2877} C_DIS
LIN {X 40.3232,Y 36.3111,Z 70,A 36.1295,B 24.8541,C -2.7869,E1 25.1175,E2 47.4765} C_DIS
LIN {X 38.0715,Y 38.6652,Z 70,A 39.4548,B 24.8536,C -2.7917,E1 25.111,E2 44.1539} C_DIS
LIN {X 36.1467,Y 40.4703,Z 70,A 41.9792,B 24.8536,C -2.7917,E1 25.1058,E2 41.6395} C_DIS
LIN {X 34.3484,Y 42.008,Z 70,A 44.8157,B 24.8524,C -2.8035,E1 25.0997,E2 38.7864} C_DIS
LIN {X 32.3457,Y 43.5692,Z 70,A 47.5406,B 24.8518,C -2.809,E1 25.0936,E2 36.0581} C_DIS
LIN {X 30.0315,Y 45.1948,Z 70,A 50.4592,B 24.8514,C -2.8125,E1 25.0869,E2 33.1412} C_DIS
LIN {X 28.0209,Y 46.4682,Z 70,A 53.1927,B 24.8505,C -2.8207,E1 25.0804,E2 30.3969} C_DIS
LIN {X 25.2049,Y 48.0536,Z 70,A 56.1489,B 24.851,C -2.816,E1 25.0732,E2 27.4602} C_DIS
LIN {X 22.2395,Y 49.4958,Z 70,A 59.8296,B 24.8502,C -2.824,E1 25.0639,E2 23.77} C_DIS
LIN {X 19.7642,Y 50.5353,Z 70,A 62.7003,B 24.8498,C -2.8276,E1 25.0564,E2 20.8974} C_DIS
LIN {X 17.2054,Y 51.4628,Z 70,A 65.53,B 24.8496,C -2.8292,E1 25.049,E2 18.0696} C_DIS
LIN {X 15.2868,Y 52.065,Z 70,A 67.6104,B 24.8496,C -2.8298,E1 25.0434,E2 15.9912} C_DIS
LIN {X 12.6127,Y 52.7768,Z 70,A 70.8371,B 24.8487,C -2.8374,E1 25.0346,E2 12.7513} C_DIS
LIN {X 8.2528,Y 53.631,Z 70,A 75.5325,B 24.8486,C -2.8392,E1 25.0217,E2 8.0569} C_DIS
LIN {X 4.5947,Y 54.0671,Z 70,A 79.5161,B 24.8483,C -2.8414,E1 25.0107,E2 4.0704} C_DIS
LIN {X 1.5023,Y 54.242,Z 70,A 83.1327,B 24.8477,C -2.8476,E1 25.0005,E2 0.4399} C_DIS
LIN {X -4.0187,Y 54.1144,Z 70,A 87.9134,B 24.8499,C -2.8263,E1 24.9873,E2 -4.2909} C_DIS
LIN {X -7.0052,Y 53.8085,Z 70,A 91.895,B 24.8485,C -2.8393,E1 24.9762,E2 -8.3061} C_DIS
LIN {X -10.2854,Y 53.2789,Z 70,A 94.5031,B 24.8505,C -2.8205,E1 24.9691,E2 -10.8721} C_DIS
LIN {X -12.2161,Y 52.8696,Z 70,A 97.0638,B 24.8498,C -2.8272,E1 24.9621,E2 -13.4519} C_DIS
LIN {X -15.0064,Y 52.1468,Z 70,A 100.1238,B 24.8501,C -2.8244,E1 24.9539,E2 -16.5099} C_DIS
LIN {X -17.8036,Y 51.259,Z 70,A 103.2066,B 24.8506,C -2.8205,E1 24.9457,E2 -19.5891} C_DIS
LIN {X -20.1544,Y 50.3819,Z 70,A 105.8517,B 24.8509,C -2.8169,E1 24.9388,E2 -22.2313} C_DIS
LIN {X -22.7772,Y 49.2508,Z 70,A 108.7605,B 24.8516,C -2.8107,E1 24.9314,E2 -25.1322} C_DIS
LIN {X -24.7454,Y 48.2918,Z 70,A 111.3711,B 24.8514,C -2.8121,E1 24.9249,E2 -27.7533} C_DIS
LIN {X -26.9099,Y 47.1201,Z 70,A 113.5622,B 24.8526,C -2.8007,E1 24.9196,E2 -29.9236} C_DIS
LIN {X -28.2766,Y 46.3128,Z 70,A 115.7285,B 24.8521,C -2.806,E1 24.9144,E2 -32.1092} C_DIS
LIN {X -31.7593,Y 43.9985,Z 70,A 119.9465,B 24.8533,C -2.7941,E1 24.9047,E2 -36.313} C_DIS
LIN {X -33.8483,Y 42.4121,Z 70,A 123.1055,B 24.8533,C -2.7948,E1 24.8978,E2 -39.4853} C_DIS
LIN {X -36.4925,Y 40.1596,Z 70,A 126.85,B 24.854,C -2.7878,E1 24.8899,E2 -43.2281} C_DIS
LIN {X -39.0886,Y 37.6365,Z 70,A 130.229,B 24.8557,C -2.7715,E1 24.8833,E2 -46.5824} C_DIS
LIN {X -40.772,Y 35.8064,Z 70,A 133.4273,B 24.8554,C -2.7743,E1 24.8774,E2 -49.8017} C_DIS
LIN {X -43.0722,Y 33.0036,Z 70,A 136.8137,B 24.8572,C -2.7572,E1 24.8716,E2 -53.1632} C_DIS
LIN {X -44.6901,Y 30.7779,Z 70,A 139.628,B 24.8582,C -2.748,E1 24.867,E2 -55.9692} C_DIS
LIN {X -45.9198,Y 28.9109,Z 70,A 142.3527,B 24.8582,C -2.7473,E1 24.8629,E2 -58.706} C_DIS
LIN {X -48.0693,Y 25.1751,Z 70,A 146.2769,B 24.8606,C -2.7244,E1 24.8576,E2 -62.596} C_DIS
LIN {X -49.2483,Y 22.7821,Z 70,A 149.5593,B 24.8606,C -2.7235,E1 24.8537,E2 -65.8941} C_DIS
LIN {X -50.3981,Y 20.1118,Z 70,A 152.5764,B 24.8617,C -2.7135,E1 24.8504,E2 -68.904} C_DIS
LIN {X -51.4784,Y 17.1593,Z 70,A 155.8718,B 24.8628,C -2.703,E1 24.8474,E2 -72.1931} C_DIS
LIN {X -52.3107,Y 14.4255,Z 70,A 158.8175,B 24.8639,C -2.6926,E1 24.8451,E2 -75.131} C_DIS
LIN {X -52.8702,Y 12.2136,Z 70,A 161.8205,B 24.8637,C -2.6944,E1 24.8432,E2 -78.156} C_DIS
LIN {X -53.5958,Y 8.4829,Z 70,A 165.3994,B 24.8656,C -2.675,E1 24.8414,E2 -81.7096} C_DIS
LIN {X -54.1478,Y 3.5302,Z 70,A 170.6679,B 24.8673,C -2.6585,E1 24.84,E2 -86.9702} C_DIS
LIN {X -54.2638,Y -0.211,Z 70,A 174.8125,B 24.8682,C -2.649,E1 24.8398,E2 -91.1172} C_DIS
LIN {X -54.1708,Y -3.1598,Z 70,A 177.7679,B 24.8695,C -2.6368,E1 24.8402,E2 -94.0611} C_DIS
LIN {X -53.9682,Y -5.6444,Z 70,A -179.6836,B 24.8704,C -2.6273,E1 24.8408,E2 -96.6022} C_DIS
LIN {X -53.5937,Y -8.4954,Z 70,A -176.2973,B 24.8708,C -2.6234,E1 24.8422,E2 -99.9994} C_DIS
LIN {X -53.0624,Y -11.3513,Z 70,A -173.436,B 24.872,C -2.6108,E1 24.8438,E2 -102.8474} C_DIS
LIN {X -52.4859,Y -13.7745,Z 70,A -170.7899,B 24.8728,C -2.6031,E1 24.8456,E2 -105.4907} C_DIS
LIN {X -51.5156,Y -17.049,Z 70,A -166.9959,B 24.8735,C -2.5955,E1 24.8487,E2 -109.2883} C_DIS
LIN {X -50.5941,Y -19.6144,Z 70,A -164.1553,B 24.8744,C -2.5867,E1 24.8515,E2 -112.1237} C_DIS
LIN {X -49.4759,Y -22.2836,Z 70,A -161.3188,B 24.8756,C -2.5746,E1 24.8546,E2 -114.947} C_DIS
LIN {X -47.9938,Y -25.3185,Z 70,A -158.1163,B 24.8771,C -2.559,E1 24.8586,E2 -118.1296} C_DIS
LIN {X -46.9319,Y -27.2352,Z 70,A -155.2803,B 24.8768,C -2.5614,E1 24.8625,E2 -120.986} C_DIS
LIN {X -45.6438,Y -29.344,Z 70,A -152.6542,B 24.8775,C -2.555,E1 24.8664,E2 -123.6102} C_DIS
LIN {X -43.996,Y -31.7628,Z 70,A -149.4436,B 24.878,C -2.5493,E1 24.8715,E2 -126.8231} C_DIS
LIN {X -42.3299,Y -33.9512,Z 70,A -146.4987,B 24.8786,C -2.5432,E1 24.8766,E2 -129.7673} C_DIS
LIN {X -40.7085,Y -35.8791,Z 70,A -143.8537,B 24.8792,C -2.537,E1 24.8814,E2 -132.4095} C_DIS
LIN {X -38.9916,Y -37.7372,Z 70,A -141.0994,B 24.8796,C -2.5327,E1 24.8867,E2 -135.1656} C_DIS
LIN {X -36.9248,Y -39.763,Z 70,A -138.184,B 24.8804,C -2.5242,E1 24.8926,E2 -138.0726} C_DIS
LIN {X -35.0581,Y -41.4173,Z 70,A -135.5194,B 24.8808,C -2.5197,E1 24.8982,E2 -140.737} C_DIS
LIN {X -33.2095,Y -42.9135,Z 70,A -132.9379,B 24.8811,C -2.5165,E1 24.9039,E2 -143.3203} C_DIS
LIN {X -30.912,Y -44.5969,Z 70,A -130.03,B 24.8818,C -2.5098,E1 24.9105,E2 -146.2223} C_DIS
LIN {X -28.8347,Y -45.9674,Z 70,A -127.3774,B 24.8821,C -2.5063,E1 24.9167,E2 -148.8751} C_DIS
LIN {X -25.7669,Y -47.7547,Z 70,A -123.5308,B 24.8824,C -2.5029,E1 24.9261,E2 -152.7248} C_DIS
LIN {X -23.2312,Y -49.0391,Z 70,A -120.5775,B 24.8828,C -2.4985,E1 24.9335,E2 -155.6753} C_DIS
LIN {X -20.9385,Y -50.0602,Z 70,A -117.9215,B 24.8831,C -2.4958,E1 24.9403,E2 -158.3313} C_DIS
LIN {X -18.3712,Y -51.0586,Z 70,A -115.3315,B 24.8839,C -2.4875,E1 24.947,E2 -160.9067} C_DIS
LIN {X -16.93,Y -51.5544,Z 70,A -113.2708,B 24.8832,C -2.4944,E1 24.9525,E2 -162.9879} C_DIS
LIN {X -13.8721,Y -52.4603,Z 70,A -110.3774,B 24.8842,C -2.4835,E1 24.9602,E2 -165.86} C_DIS
LIN {X -11.1357,Y -53.1072,Z 70,A -106.7465,B 24.8832,C -2.4944,E1 24.9702,E2 -169.5214} C_DIS
LIN {X -7.5519,Y -53.7346,Z 70,A -102.8312,B 24.8832,C -2.4948,E1 24.981,E2 -173.4411} C_DIS
LIN {X -4.1389,Y -54.1042,Z 70,A -99.2506,B 24.8832,C -2.4938,E1 24.991,E2 -177.021} C_DIS
LIN {X 0.046,Y -54.2633,Z 70,A -95.0645,B 24.8836,C -2.4899,E1 25.0026,E2 -181.1983} C_DIS
LIN {X 0.046,Y -54.2633,Z 70,A -95.0645,B 24.8836,C -2.4899,E1 25.0026,E2 -181.1983} C_DIS
Enddeposition()
LIN {X 0.2727,Y -53.3094,Z 70,A -95.1906,B 24.8827,C -2.4993,E1 25.0024,E2 -181.0945} C_DIS
Startdeposition()
$VEL.CP = VEL_PRINT
LIN {X -2.7183,Y -53.2423,Z 70,A -99.4497,B 24.8846,C -2.4794,E1 24.9903,E2 -176.7877} C_DIS
LIN {X -4.8561,Y -53.0896,Z 70,A -101.7826,B 24.8846,C -2.4789,E1 24.9838,E2 -174.4526} C_DIS
LIN {X -7.2548,Y -52.8158,Z 70,A -104.4068,B 24.8846,C -2.4789,E1 24.9766,E2 -171.8264} C_DIS
LIN {X -9.8138,Y -52.4008,Z 70,A -107.1703,B 24.8846,C -2.4801,E1 24.969,E2 -169.0631} C_DIS
LIN {X -12.2373,Y -51.8882,Z 70,A -109.8791,B 24.8846,C -2.4805,E1 24.9616,E2 -166.3519} C_DIS
LIN {X -14.8727,Y -51.1955,Z 70,A -112.7435,B 24.8842,C -2.4835,E1 24.9539,E2 -163.49} C_DIS
LIN {X -17.3578,Y -50.4072,Z 70,A -115.5555,B 24.884,C -2.4855,E1 24.9464,E2 -160.6776} C_DIS
LIN {X -19.8022,Y -49.498,Z 70,A -118.3853,B 24.8839,C -2.4876,E1 24.939,E2 -157.8468} C_DIS
LIN {X -22.2001,Y -48.47,Z 70,A -121.183,B 24.8836,C -2.4907,E1 24.9319,E2 -155.0498} C_DIS
LIN {X -24.4545,Y -47.372,Z 70,A -123.9464,B 24.8834,C -2.4928,E1 24.925,E2 -152.284} C_DIS
LIN {X -26.8294,Y -46.0691,Z 70,A -126.8525,B 24.883,C -2.4968,E1 24.9179,E2 -149.379} C_DIS
LIN {X -29.0822,Y -44.6812,Z 70,A -129.655,B 24.8825,C -2.5017,E1 24.9113,E2 -146.5793} C_DIS
LIN {X -31.1533,Y -43.2621,Z 70,A -132.3973,B 24.8822,C -2.5054,E1 24.9051,E2 -143.8365} C_DIS
LIN {X -33.2742,Y -41.6532,Z 70,A -135.2847,B 24.8817,C -2.51,E1 24.8987,E2 -140.9494} C_DIS
LIN {X -35.2742,Y -39.9736,Z 70,A -138.0894,B 24.8812,C -2.5153,E1 24.8928,E2 -138.1465} C_DIS
LIN {X -37.2257,Y -38.1631,Z 70,A -140.9637,B 24.8807,C -2.5209,E1 24.8869,E2 -135.2735} C_DIS
LIN {X -39.0673,Y -36.2757,Z 70,A -143.8105,B 24.8802,C -2.5267,E1 24.8815,E2 -132.4282} C_DIS
LIN {X -40.764,Y -34.3578,Z 70,A -146.5948,B 24.8796,C -2.5323,E1 24.8764,E2 -129.6448} C_DIS
LIN {X -42.4289,Y -32.2796,Z 70,A -149.4549,B 24.879,C -2.5391,E1 24.8715,E2 -126.7873} C_DIS
LIN {X -43.9961,Y -30.108,Z 70,A -152.2891,B 24.8782,C -2.5468,E1 24.8669,E2 -123.9577} C_DIS
LIN {X -45.4033,Y -27.9411,Z 70,A -155.1353,B 24.8777,C -2.5528,E1 24.8627,E2 -121.1114} C_DIS
LIN {X -46.6599,Y -25.7874,Z 70,A -157.8689,B 24.8771,C -2.559,E1 24.8589,E2 -118.3783} C_DIS
LIN {X -47.8602,Y -23.4847,Z 70,A -160.6901,B 24.8764,C -2.5661,E1 24.8553,E2 -115.559} C_DIS
LIN {X -49.0014,Y -21.0012,Z 70,A -163.5766,B 24.8755,C -2.5751,E1 24.8521,E2 -112.678} C_DIS
LIN {X -49.9711,Y -18.5762,Z 70,A -166.4096,B 24.8748,C -2.5827,E1 24.8492,E2 -109.8473} C_DIS
LIN {X -50.8275,Y -16.0853,Z 70,A -169.2777,B 24.874,C -2.5904,E1 24.8467,E2 -106.9813} C_DIS
LIN {X -51.5271,Y -13.6781,Z 70,A -171.9926,B 24.8733,C -2.5981,E1 24.8447,E2 -104.269} C_DIS
LIN {X -52.1346,Y -11.1409,Z 70,A -174.8485,B 24.8725,C -2.6058,E1 24.8429,E2 -101.4148} C_DIS
LIN {X -52.6381,Y -8.4499,Z 70,A -177.7417,B 24.8716,C -2.6156,E1 24.8415,E2 -98.5277} C_DIS
LIN {X -52.9767,Y -5.9667,Z 70,A 179.4736,B 24.8709,C -2.6226,E1 24.8406,E2 -95.7431} C_DIS
LIN {X -53.2051,Y -3.3683,Z 70,A 176.6838,B 24.87,C -2.6315,E1 24.84,E2 -92.9579} C_DIS
LIN {X -53.308,Y -0.6601,Z 70,A 173.866,B 24.8689,C -2.6421,E1 24.8398,E2 -90.1484} C_DIS
LIN {X -53.279,Y 1.8656,Z 70,A 170.984,B 24.8683,C -2.6482,E1 24.84,E2 -87.2636} C_DIS
LIN {X -53.1136,Y 4.5951,Z 70,A 168.0591,B 24.8674,C -2.6576,E1 24.8406,E2 -84.3437} C_DIS
LIN {X -52.8392,Y 7.0819,Z 70,A 165.3148,B 24.8666,C -2.6653,E1 24.8415,E2 -81.6013} C_DIS
LIN {X -52.4123,Y 9.7535,Z 70,A 162.4177,B 24.8657,C -2.6745,E1 24.8429,E2 -78.7092} C_DIS
LIN {X -51.8907,Y 12.2267,Z 70,A 159.6467,B 24.8649,C -2.6822,E1 24.8445,E2 -75.9402} C_DIS
LIN {X -51.2019,Y 14.8511,Z 70,A 156.7734,B 24.8639,C -2.6918,E1 24.8467,E2 -73.0732} C_DIS
LIN {X -50.4129,Y 17.3414,Z 70,A 153.9212,B 24.8631,C -2.6997,E1 24.8492,E2 -70.2237} C_DIS
LIN {X -49.4819,Y 19.8417,Z 70,A 151.0404,B 24.8623,C -2.7082,E1 24.8521,E2 -67.3468} C_DIS
LIN {X -48.461,Y 22.2195,Z 70,A 148.2863,B 24.8614,C -2.7168,E1 24.8552,E2 -64.5982} C_DIS
LIN {X -47.3677,Y 24.463,Z 70,A 145.4985,B 24.8607,C -2.723,E1 24.8586,E2 -61.8103} C_DIS
LIN {X -46.07,Y 26.8277,Z 70,A 142.6376,B 24.8598,C -2.7318,E1 24.8626,E2 -58.9554} C_DIS
LIN {X -44.6871,Y 29.0732,Z 70,A 139.7867,B 24.8591,C -2.7394,E1 24.8668,E2 -56.1081} C_DIS
LIN {X -43.2694,Y 31.143,Z 70,A 137.0449,B 24.8584,C -2.7459,E1 24.8712,E2 -53.3686} C_DIS
LIN {X -41.6541,Y 33.2731,Z 70,A 134.1271,B 24.8577,C -2.7527,E1 24.8762,E2 -50.4532} C_DIS
LIN {X -39.9654,Y 35.2836,Z 70,A 131.3163,B 24.8569,C -2.76,E1 24.8813,E2 -47.647} C_DIS
LIN {X -38.1581,Y 37.231,Z 70,A 128.4446,B 24.8562,C -2.7666,E1 24.8868,E2 -44.7787} C_DIS
LIN {X -36.3355,Y 39.0112,Z 70,A 125.6689,B 24.8556,C -2.7724,E1 24.8924,E2 -42.0052} C_DIS
LIN {X -34.3525,Y 40.7685,Z 70,A 122.8196,B 24.855,C -2.7787,E1 24.8985,E2 -39.1598} C_DIS
LIN {X -32.2773,Y 42.4307,Z 70,A 119.9885,B 24.8543,C -2.785,E1 24.9047,E2 -36.3336} C_DIS
LIN {X -30.2194,Y 43.9197,Z 70,A 117.5646,B 24.8532,C -2.7953,E1 24.9101,E2 -33.9258} C_DIS
LIN {X -28.5233,Y 45.0401,Z 70,A 115.0361,B 24.8534,C -2.7939,E1 24.9161,E2 -31.3857} C_DIS
LIN {X -26.3882,Y 46.3226,Z 70,A 112.3161,B 24.8529,C -2.7979,E1 24.9227,E2 -28.6671} C_DIS
LIN {X -23.9564,Y 47.6264,Z 70,A 109.3573,B 24.8524,C -2.8028,E1 24.93,E2 -25.7119} C_DIS
LIN {X -21.6883,Y 48.7007,Z 70,A 106.6497,B 24.852,C -2.8067,E1 24.9368,E2 -23.0068} C_DIS
Enddeposition()
END
